TEXTLIST S1_Prompts
  0 = 'Waiting for Station 1 Clamp A1 Advance... Check Q1.0...' | German: 'S1_Prompts German 0' | French: 'S1_Prompts French 0' | 汉语: '汉语'
  1 = 'Waiting for Station 1 Clamp A1 Return... Check Q1.1...' | German: 'S1_Prompts German 1' | French: 'S1_Prompts French 1' | 汉语: '汉语'
  2 = 'Spare' | German: 'S1_Prompts German 2' | French: 'S1_Prompts French 2' | 汉语: '汉语'
  3 = 'Spare' | German: 'S1_Prompts German 3' | French: 'S1_Prompts French 3'
  4 = 'Spare' | German: 'S1_Prompts German 4' | French: 'S1_Prompts French 4'
  5 = 'Spare' | German: 'S1_Prompts German 5' | French: 'S1_Prompts French 5'
  6 = 'Spare' | German: 'S1_Prompts German 6' | French: 'S1_Prompts French 6'
  7 = 'Spare' | German: 'S1_Prompts German 7' | French: 'S1_Prompts French 7'
  8 = 'Spare' | German: 'S1_Prompts German 8' | French: 'S1_Prompts French 8'
  9 = 'Spare' | German: 'S1_Prompts German 9' | French: 'S1_Prompts French 9'
  10 = 'Waiting for Lock Cylinder A2 Lock... Check Q1.2...' | German: 'S1_Prompts German 10' | French: 'S1_Prompts French 10'
  11 = 'Waiting for Lock Cylinder A2 Unlock... Check Q1.3...' | German: 'S1_Prompts German 11' | French: 'S1_Prompts French 11'
  12 = 'Spare' | German: 'S1_Prompts German 12' | French: 'S1_Prompts French 12'
  13 = 'Spare' | German: 'S1_Prompts German 13' | French: 'S1_Prompts French 13'
  14 = 'Spare' | German: 'S1_Prompts German 14' | French: 'S1_Prompts French 14'
  15 = 'Spare' | German: 'S1_Prompts German 15' | French: 'S1_Prompts French 15'
  16 = 'Spare' | German: 'S1_Prompts German 16' | French: 'S1_Prompts French 16'
  17 = 'Spare' | German: 'S1_Prompts German 17' | French: 'S1_Prompts French 17'
  18 = 'Spare' | German: 'S1_Prompts German 18' | French: 'S1_Prompts French 18'
  19 = 'Spare' | German: 'S1_Prompts German 19' | French: 'S1_Prompts French 19'
  20 = 'Waiting for Urger Cylinder A3 Urge... Check Q1.4...' | German: 'S1_Prompts German 20' | French: 'S1_Prompts French 20'
  21 = 'Waiting for Urger Cylinder A3 Return... Check Q1.5...' | German: 'S1_Prompts German 21' | French: 'S1_Prompts French 21'
  22 = 'Spare' | German: 'S1_Prompts German 22' | French: 'S1_Prompts French 22'
  23 = 'Spare' | German: 'S1_Prompts German 23' | French: 'S1_Prompts French 23'
  24 = 'Spare' | German: 'S1_Prompts German 24' | French: 'S1_Prompts French 24'
  25 = 'Spare' | German: 'S1_Prompts German 25' | French: 'S1_Prompts French 25'
  26 = 'Spare' | German: 'S1_Prompts German 26' | French: 'S1_Prompts French 26'
  27 = 'Spare' | German: 'S1_Prompts German 27' | French: 'S1_Prompts French 27'
  28 = 'Spare' | German: 'S1_Prompts German 28' | French: 'S1_Prompts French 28'
  29 = 'Spare' | German: 'S1_Prompts German 29' | French: 'S1_Prompts French 29'
  30 = 'Waiting for Clamp Cylinder A1 Advance... Check Q1.0...' | German: 'S1_Prompts German 30' | French: 'S1_Prompts French 30'
  31 = 'Waiting for Clamp Cylinder A1 Return... Check Q1.1...' | German: 'S1_Prompts German 31' | French: 'S1_Prompts French 31'
  32 = 'Spare' | German: 'S1_Prompts German 32' | French: 'S1_Prompts French 32'
  33 = 'Spare' | German: 'S1_Prompts German 33' | French: 'S1_Prompts French 33'
  34 = 'Spare' | German: 'S1_Prompts German 34' | French: 'S1_Prompts French 34'
  35 = 'Spare' | German: 'S1_Prompts German 35' | French: 'S1_Prompts French 35'
  36 = 'Spare' | German: 'S1_Prompts German 36' | French: 'S1_Prompts French 36'
  37 = 'Spare' | German: 'S1_Prompts German 37' | French: 'S1_Prompts French 37'
  38 = 'Spare' | German: 'S1_Prompts German 38' | French: 'S1_Prompts French 38'
  39 = 'Spare' | German: 'S1_Prompts German 39' | French: 'S1_Prompts French 39'
  40 = 'Waiting for Clamp Cylinder A1 Advance... Check Q1.0...' | German: 'S1_Prompts German 40' | French: 'S1_Prompts French 40'
  41 = 'Waiting for Clamp Cylinder A1 Return... Check Q1.1...' | German: 'S1_Prompts German 41' | French: 'S1_Prompts French 41'
  42 = 'Spare' | German: 'S1_Prompts German 42' | French: 'S1_Prompts French 42'
  43 = 'Spare' | German: 'S1_Prompts German 43' | French: 'S1_Prompts French 43'
  44 = 'Spare' | German: 'S1_Prompts German 44' | French: 'S1_Prompts French 44'
  45 = 'Spare' | German: 'S1_Prompts German 45' | French: 'S1_Prompts French 45'
  46 = 'Spare' | German: 'S1_Prompts German 46' | French: 'S1_Prompts French 46'
  47 = 'Spare' | German: 'S1_Prompts German 47' | French: 'S1_Prompts French 47'
  48 = 'Spare' | German: 'S1_Prompts German 48' | French: 'S1_Prompts French 48'
  49 = 'Spare' | German: 'S1_Prompts German 49' | French: 'S1_Prompts French 49'
  50 = 'Waiting for Clamp Cylinder A1 Advance... Check Q1.0...' | German: 'S1_Prompts German 50' | French: 'S1_Prompts French 50'
  51 = 'Waiting for Clamp Cylinder A1 Return... Check Q1.1...' | German: 'S1_Prompts German 51' | French: 'S1_Prompts French 51'
  52 = 'Spare' | German: 'S1_Prompts German 52' | French: 'S1_Prompts French 52'
  53 = 'Spare' | German: 'S1_Prompts German 53' | French: 'S1_Prompts French 53'
  54 = 'Spare' | German: 'S1_Prompts German 54' | French: 'S1_Prompts French 54'
  55 = 'Spare' | German: 'S1_Prompts German 55' | French: 'S1_Prompts French 55'
  56 = 'Spare' | German: 'S1_Prompts German 56' | French: 'S1_Prompts French 56'
  57 = 'Spare' | German: 'S1_Prompts German 57' | French: 'S1_Prompts French 57'
  58 = 'Spare' | German: 'S1_Prompts German 58' | French: 'S1_Prompts French 58'
  59 = 'Spare' | German: 'S1_Prompts German 59' | French: 'S1_Prompts French 59'
  60 = 'Waiting for Clamp Cylinder A1 Advance... Check Q1.0...' | German: 'S1_Prompts German 60' | French: 'S1_Prompts French 60'
  61 = 'Waiting for Clamp Cylinder A1 Return... Check Q1.1...' | German: 'S1_Prompts German 61' | French: 'S1_Prompts French 61'
  62 = 'Spare' | German: 'S1_Prompts German 62' | French: 'S1_Prompts French 62'
  63 = 'Spare' | German: 'S1_Prompts German 63' | French: 'S1_Prompts French 63'
  64 = 'Spare' | German: 'S1_Prompts German 64' | French: 'S1_Prompts French 64'
  65 = 'Spare' | German: 'S1_Prompts German 65' | French: 'S1_Prompts French 65'
  66 = 'Spare' | German: 'S1_Prompts German 66' | French: 'S1_Prompts French 66'
  67 = 'Spare' | German: 'S1_Prompts German 67' | French: 'S1_Prompts French 67'
  68 = 'Spare' | German: 'S1_Prompts German 68' | French: 'S1_Prompts French 68'
  69 = 'Spare' | German: 'S1_Prompts German 69' | French: 'S1_Prompts French 69'
  70 = 'Waiting for Clamp Cylinder A1 Advance... Check Q1.0...' | German: 'S1_Prompts German 70' | French: 'S1_Prompts French 70'
  71 = 'Waiting for Clamp Cylinder A1 Return... Check Q1.1...' | German: 'S1_Prompts German 71' | French: 'S1_Prompts French 71'
  72 = 'Spare' | German: 'S1_Prompts German 72' | French: 'S1_Prompts French 72'
  73 = 'Spare' | German: 'S1_Prompts German 73' | French: 'S1_Prompts French 73'
  74 = 'Spare' | German: 'S1_Prompts German 74' | French: 'S1_Prompts French 74'
  75 = 'Spare' | German: 'S1_Prompts German 75' | French: 'S1_Prompts French 75'
  76 = 'Spare' | German: 'S1_Prompts German 76' | French: 'S1_Prompts French 76'
  77 = 'Spare' | German: 'S1_Prompts German 77' | French: 'S1_Prompts French 77'
  78 = 'Spare' | German: 'S1_Prompts German 78' | French: 'S1_Prompts French 78'
  79 = 'Spare' | German: 'S1_Prompts German 79' | French: 'S1_Prompts French 79'
  80 = 'Waiting for Clamp Cylinder A1 Advance... Check Q1.0...' | German: 'S1_Prompts German 80' | French: 'S1_Prompts French 80'
  81 = 'Waiting for Clamp Cylinder A1 Return... Check Q1.1...' | German: 'S1_Prompts German 81' | French: 'S1_Prompts French 81'
  82 = 'Spare' | German: 'S1_Prompts German 82' | French: 'S1_Prompts French 82'
  83 = 'Spare' | German: 'S1_Prompts German 83' | French: 'S1_Prompts French 83'
  84 = 'Spare' | German: 'S1_Prompts German 84' | French: 'S1_Prompts French 84'
  85 = 'Spare' | German: 'S1_Prompts German 85' | French: 'S1_Prompts French 85'
  86 = 'Spare' | German: 'S1_Prompts German 86' | French: 'S1_Prompts French 86'
  87 = 'Spare' | German: 'S1_Prompts German 87' | French: 'S1_Prompts French 87'
  88 = 'Spare' | German: 'S1_Prompts German 88' | French: 'S1_Prompts French 88'
  89 = 'Spare' | German: 'S1_Prompts German 89' | French: 'S1_Prompts French 89'
  90 = 'Waiting for Clamp Cylinder A1 Advance... Check Q1.0...' | German: 'S1_Prompts German 90' | French: 'S1_Prompts French 90'
  91 = 'Waiting for Clamp Cylinder A1 Return... Check Q1.1...' | German: 'S1_Prompts German 91' | French: 'S1_Prompts French 91'
  92 = 'Spare' | German: 'S1_Prompts German 92' | French: 'S1_Prompts French 92'
  93 = 'Spare' | German: 'S1_Prompts German 93' | French: 'S1_Prompts French 93'
  94 = 'Spare' | German: 'S1_Prompts German 94' | French: 'S1_Prompts French 94'
  95 = 'Spare' | German: 'S1_Prompts German 95' | French: 'S1_Prompts French 95'
  96 = 'Spare' | German: 'S1_Prompts German 96' | French: 'S1_Prompts French 96'
  97 = 'Spare' | German: 'S1_Prompts German 97' | French: 'S1_Prompts French 97'
  98 = 'Spare' | German: 'S1_Prompts German 98' | French: 'S1_Prompts French 98'
  99 = 'Spare' | German: 'S1_Prompts German 99' | French: 'S1_Prompts French 99'
  100 = 'Waiting for Clamp Cylinder A1 Advance... Check Q1.0...' | German: 'S1_Prompts German 100' | French: 'S1_Prompts French 100'
  101 = 'Waiting for Clamp Cylinder A1 Return... Check Q1.1...' | German: 'S1_Prompts German 101' | French: 'S1_Prompts French 101'
  102 = 'Spare' | German: 'S1_Prompts German 102' | French: 'S1_Prompts French 102'
  103 = 'Spare' | German: 'S1_Prompts German 103' | French: 'S1_Prompts French 103'
  104 = 'Spare' | German: 'S1_Prompts German 104' | French: 'S1_Prompts French 104'
  105 = 'Spare' | German: 'S1_Prompts German 105' | French: 'S1_Prompts French 105'
  106 = 'Spare' | German: 'S1_Prompts German 106' | French: 'S1_Prompts French 106'
  107 = 'Spare' | German: 'S1_Prompts German 107' | French: 'S1_Prompts French 107'
  108 = 'Spare' | German: 'S1_Prompts German 108' | French: 'S1_Prompts French 108'
  109 = 'Spare' | German: 'S1_Prompts German 109' | French: 'S1_Prompts French 109'
  110 = 'Waiting for Clamp Cylinder A1 Advance... Check Q1.0...' | German: 'S1_Prompts German 110' | French: 'S1_Prompts French 110'
  111 = 'Waiting for Clamp Cylinder A1 Return... Check Q1.1...' | German: 'S1_Prompts German 111' | French: 'S1_Prompts French 111'
  112 = 'Spare' | German: 'S1_Prompts German 112' | French: 'S1_Prompts French 112'
  113 = 'Spare' | German: 'S1_Prompts German 113' | French: 'S1_Prompts French 113'
  114 = 'Spare' | German: 'S1_Prompts German 114' | French: 'S1_Prompts French 114'
  115 = 'Spare' | German: 'S1_Prompts German 115' | French: 'S1_Prompts French 115'
  116 = 'Spare' | German: 'S1_Prompts German 116' | French: 'S1_Prompts French 116'
  117 = 'Spare' | German: 'S1_Prompts German 117' | French: 'S1_Prompts French 117'
  118 = 'Spare' | German: 'S1_Prompts German 118' | French: 'S1_Prompts French 118'
  119 = 'Spare' | German: 'S1_Prompts German 119' | French: 'S1_Prompts French 119'
  120 = 'Waiting for Clamp Cylinder A1 Advance... Check Q1.0...' | German: 'S1_Prompts German 120' | French: 'S1_Prompts French 120'
  121 = 'Waiting for Clamp Cylinder A1 Return... Check Q1.1...' | German: 'S1_Prompts German 121' | French: 'S1_Prompts French 121'
  122 = 'Spare' | German: 'S1_Prompts German 122' | French: 'S1_Prompts French 122'
  123 = 'Spare' | German: 'S1_Prompts German 123' | French: 'S1_Prompts French 123'
  124 = 'Spare' | German: 'S1_Prompts German 124' | French: 'S1_Prompts French 124'
  125 = 'Spare' | German: 'S1_Prompts German 125' | French: 'S1_Prompts French 125'
  126 = 'Spare' | German: 'S1_Prompts German 126' | French: 'S1_Prompts French 126'
  127 = 'Spare' | German: 'S1_Prompts German 127' | French: 'S1_Prompts French 127'
  128 = 'Spare' | German: 'S1_Prompts German 128' | French: 'S1_Prompts French 128'
  129 = 'Spare' | German: 'S1_Prompts German 129' | French: 'S1_Prompts French 129'
  130 = 'Waiting for Clamp Cylinder A1 Advance... Check Q1.0...' | German: 'S1_Prompts German 130' | French: 'S1_Prompts French 130'
  131 = 'Waiting for Clamp Cylinder A1 Return... Check Q1.1...' | German: 'S1_Prompts German 131' | French: 'S1_Prompts French 131'
  132 = 'Spare' | German: 'S1_Prompts German 132' | French: 'S1_Prompts French 132'
  133 = 'Spare' | German: 'S1_Prompts German 133' | French: 'S1_Prompts French 133'
  134 = 'Spare' | German: 'S1_Prompts German 134' | French: 'S1_Prompts French 134'
  135 = 'Spare' | German: 'S1_Prompts German 135' | French: 'S1_Prompts French 135'
  136 = 'Spare' | German: 'S1_Prompts German 136' | French: 'S1_Prompts French 136'
  137 = 'Spare' | German: 'S1_Prompts German 137' | French: 'S1_Prompts French 137'
  138 = 'Spare' | German: 'S1_Prompts German 138' | French: 'S1_Prompts French 138'
  139 = 'Spare' | German: 'S1_Prompts German 139' | French: 'S1_Prompts French 139'
  140 = 'Waiting for Clamp Cylinder A1 Advance... Check Q1.0...' | German: 'S1_Prompts German 140' | French: 'S1_Prompts French 140'
  141 = 'Waiting for Clamp Cylinder A1 Return... Check Q1.1...' | German: 'S1_Prompts German 141' | French: 'S1_Prompts French 141'
  142 = 'Spare' | German: 'S1_Prompts German 142' | French: 'S1_Prompts French 142'
  143 = 'Spare' | German: 'S1_Prompts German 143' | French: 'S1_Prompts French 143'
  144 = 'Spare' | German: 'S1_Prompts German 144' | French: 'S1_Prompts French 144'
  145 = 'Spare' | German: 'S1_Prompts German 145' | French: 'S1_Prompts French 145'
  146 = 'Spare' | German: 'S1_Prompts German 146' | French: 'S1_Prompts French 146'
  147 = 'Spare' | German: 'S1_Prompts German 147' | French: 'S1_Prompts French 147'
  148 = 'Spare' | German: 'S1_Prompts German 148' | French: 'S1_Prompts French 148'
  149 = 'Spare' | German: 'S1_Prompts German 149' | French: 'S1_Prompts French 149'
  150 = 'Waiting for Clamp Cylinder A1 Advance... Check Q1.0...' | German: 'S1_Prompts German 150' | French: 'S1_Prompts French 150'
  151 = 'Waiting for Clamp Cylinder A1 Return... Check Q1.1...' | German: 'S1_Prompts German 151' | French: 'S1_Prompts French 151'
  152 = 'Spare' | German: 'S1_Prompts German 152' | French: 'S1_Prompts French 152'
  153 = 'Spare' | German: 'S1_Prompts German 153' | French: 'S1_Prompts French 153'
  154 = 'Spare' | German: 'S1_Prompts German 154' | French: 'S1_Prompts French 154'
  155 = 'Spare' | German: 'S1_Prompts German 155' | French: 'S1_Prompts French 155'
  156 = 'Spare' | German: 'S1_Prompts German 156' | French: 'S1_Prompts French 156'
  157 = 'Spare' | German: 'S1_Prompts German 157' | French: 'S1_Prompts French 157'
  158 = 'Spare' | German: 'S1_Prompts German 158' | French: 'S1_Prompts French 158'
  159 = 'Spare' | German: 'S1_Prompts German 159' | French: 'S1_Prompts French 159'
  160 = 'Waiting for Clamp Cylinder A1 Advance... Check Q1.0...' | German: 'S1_Prompts German 160' | French: 'S1_Prompts French 160'
  161 = 'Waiting for Clamp Cylinder A1 Return... Check Q1.1...' | German: 'S1_Prompts German 161' | French: 'S1_Prompts French 161'
  162 = 'Spare' | German: 'S1_Prompts German 162' | French: 'S1_Prompts French 162'
  163 = 'Spare' | German: 'S1_Prompts German 163' | French: 'S1_Prompts French 163'
  164 = 'Spare' | German: 'S1_Prompts German 164' | French: 'S1_Prompts French 164'
  165 = 'Spare' | German: 'S1_Prompts German 165' | French: 'S1_Prompts French 165'
  166 = 'Spare' | German: 'S1_Prompts German 166' | French: 'S1_Prompts French 166'
  167 = 'Spare' | German: 'S1_Prompts German 167' | French: 'S1_Prompts French 167'
  168 = 'Spare' | German: 'S1_Prompts German 168' | French: 'S1_Prompts French 168'
  169 = 'Spare' | German: 'S1_Prompts German 169' | French: 'S1_Prompts French 169'
  170 = 'Waiting for Clamp Cylinder A1 Advance... Check Q1.0...' | German: 'S1_Prompts German 170' | French: 'S1_Prompts French 170'
  171 = 'Waiting for Clamp Cylinder A1 Return... Check Q1.1...' | German: 'S1_Prompts German 171' | French: 'S1_Prompts French 171'
  172 = 'Spare' | German: 'S1_Prompts German 172' | French: 'S1_Prompts French 172'
  173 = 'Spare' | German: 'S1_Prompts German 173' | French: 'S1_Prompts French 173'
  174 = 'Spare' | German: 'S1_Prompts German 174' | French: 'S1_Prompts French 174'
  175 = 'Spare' | German: 'S1_Prompts German 175' | French: 'S1_Prompts French 175'
  176 = 'Spare' | German: 'S1_Prompts German 176' | French: 'S1_Prompts French 176'
  177 = 'Spare' | German: 'S1_Prompts German 177' | French: 'S1_Prompts French 177'
  178 = 'Spare' | German: 'S1_Prompts German 178' | French: 'S1_Prompts French 178'
  179 = 'Spare' | German: 'S1_Prompts German 179' | French: 'S1_Prompts French 179'
  180 = 'Waiting for Clamp Cylinder A1 Advance... Check Q1.0...' | German: 'S1_Prompts German 180' | French: 'S1_Prompts French 180'
  181 = 'Waiting for Clamp Cylinder A1 Return... Check Q1.1...' | German: 'S1_Prompts German 181' | French: 'S1_Prompts French 181'
  182 = 'Spare' | German: 'S1_Prompts German 182' | French: 'S1_Prompts French 182'
  183 = 'Spare' | German: 'S1_Prompts German 183' | French: 'S1_Prompts French 183'
  184 = 'Spare' | German: 'S1_Prompts German 184' | French: 'S1_Prompts French 184'
  185 = 'Spare' | German: 'S1_Prompts German 185' | French: 'S1_Prompts French 185'
  186 = 'Spare' | German: 'S1_Prompts German 186' | French: 'S1_Prompts French 186'
  187 = 'Spare' | German: 'S1_Prompts German 187' | French: 'S1_Prompts French 187'
  188 = 'Spare' | German: 'S1_Prompts German 188' | French: 'S1_Prompts French 188'
  189 = 'Spare' | German: 'S1_Prompts German 189' | French: 'S1_Prompts French 189'
  190 = 'Waiting for Clamp Cylinder A1 Advance... Check Q1.0...' | German: 'S1_Prompts German 190' | French: 'S1_Prompts French 190'
  191 = 'Waiting for Clamp Cylinder A1 Return... Check Q1.1...' | German: 'S1_Prompts German 191' | French: 'S1_Prompts French 191'
  192 = 'Spare' | German: 'S1_Prompts German 192' | French: 'S1_Prompts French 192'
  193 = 'Spare' | German: 'S1_Prompts German 193' | French: 'S1_Prompts French 193'
  194 = 'Spare' | German: 'S1_Prompts German 194' | French: 'S1_Prompts French 194'
  195 = 'Spare' | German: 'S1_Prompts German 195' | French: 'S1_Prompts French 195'
  196 = 'Spare' | German: 'S1_Prompts German 196' | French: 'S1_Prompts French 196'
  197 = 'Spare' | German: 'S1_Prompts German 197' | French: 'S1_Prompts French 197'
  198 = 'Spare' | German: 'S1_Prompts German 198' | French: 'S1_Prompts French 198'
  199 = 'Spare' | German: 'S1_Prompts German 199' | French: 'S1_Prompts French 199'
  200 = 'Waiting for Clamp Cylinder A1 Advance... Check Q1.0...' | German: 'S1_Prompts German 200' | French: 'S1_Prompts French 200'
  201 = 'Waiting for Clamp Cylinder A1 Return... Check Q1.1...' | German: 'S1_Prompts German 201' | French: 'S1_Prompts French 201'
  202 = 'Spare' | German: 'S1_Prompts German 202' | French: 'S1_Prompts French 202'
  203 = 'Spare' | German: 'S1_Prompts German 203' | French: 'S1_Prompts French 203'
  204 = 'Spare' | German: 'S1_Prompts German 204' | French: 'S1_Prompts French 204'
  205 = 'Spare' | German: 'S1_Prompts German 205' | French: 'S1_Prompts French 205'
  206 = 'Spare' | German: 'S1_Prompts German 206' | French: 'S1_Prompts French 206'
  207 = 'Spare' | German: 'S1_Prompts German 207' | French: 'S1_Prompts French 207'
  208 = 'Spare' | German: 'S1_Prompts German 208' | French: 'S1_Prompts French 208'
  209 = 'Spare' | German: 'S1_Prompts German 209' | French: 'S1_Prompts French 209'
  210 = 'Waiting for Clamp Cylinder A1 Advance... Check Q1.0...' | German: 'S1_Prompts German 210' | French: 'S1_Prompts French 210'
  211 = 'Waiting for Clamp Cylinder A1 Return... Check Q1.1...' | German: 'S1_Prompts German 211' | French: 'S1_Prompts French 211'
  212 = 'Spare' | German: 'S1_Prompts German 212' | French: 'S1_Prompts French 212'
  213 = 'Spare' | German: 'S1_Prompts German 213' | French: 'S1_Prompts French 213'
  214 = 'Spare' | German: 'S1_Prompts German 214' | French: 'S1_Prompts French 214'
  215 = 'Spare' | German: 'S1_Prompts German 215' | French: 'S1_Prompts French 215'
  216 = 'Spare' | German: 'S1_Prompts German 216' | French: 'S1_Prompts French 216'
  217 = 'Spare' | German: 'S1_Prompts German 217' | French: 'S1_Prompts French 217'
  218 = 'Spare' | German: 'S1_Prompts German 218' | French: 'S1_Prompts French 218'
  219 = 'Spare' | German: 'S1_Prompts German 219' | French: 'S1_Prompts French 219'
  220 = 'Waiting for Clamp Cylinder A1 Advance... Check Q1.0...' | German: 'S1_Prompts German 220' | French: 'S1_Prompts French 220'
  221 = 'Waiting for Clamp Cylinder A1 Return... Check Q1.1...' | German: 'S1_Prompts German 221' | French: 'S1_Prompts French 221'
  222 = 'Spare' | German: 'S1_Prompts German 222' | French: 'S1_Prompts French 222'
  223 = 'Spare' | German: 'S1_Prompts German 223' | French: 'S1_Prompts French 223'
  224 = 'Spare' | German: 'S1_Prompts German 224' | French: 'S1_Prompts French 224'
  225 = 'Spare' | German: 'S1_Prompts German 225' | French: 'S1_Prompts French 225'
  226 = 'Spare' | German: 'S1_Prompts German 226' | French: 'S1_Prompts French 226'
  227 = 'Spare' | German: 'S1_Prompts German 227' | French: 'S1_Prompts French 227'
  228 = 'Spare' | German: 'S1_Prompts German 228' | French: 'S1_Prompts French 228'
  229 = 'Spare' | German: 'S1_Prompts German 229' | French: 'S1_Prompts French 229'
  230 = 'Waiting for Clamp Cylinder A1 Advance... Check Q1.0...' | German: 'S1_Prompts German 230' | French: 'S1_Prompts French 230'
  231 = 'Waiting for Clamp Cylinder A1 Return... Check Q1.1...' | German: 'S1_Prompts German 231' | French: 'S1_Prompts French 231'
  232 = 'Spare' | German: 'S1_Prompts German 232' | French: 'S1_Prompts French 232'
  233 = 'Spare' | German: 'S1_Prompts German 233' | French: 'S1_Prompts French 233'
  234 = 'Spare' | German: 'S1_Prompts German 234' | French: 'S1_Prompts French 234'
  235 = 'Spare' | German: 'S1_Prompts German 235' | French: 'S1_Prompts French 235'
  236 = 'Spare' | German: 'S1_Prompts German 236' | French: 'S1_Prompts French 236'
  237 = 'Spare' | German: 'S1_Prompts German 237' | French: 'S1_Prompts French 237'
  238 = 'Spare' | German: 'S1_Prompts German 238' | French: 'S1_Prompts French 238'
  239 = 'Spare' | German: 'S1_Prompts German 239' | French: 'S1_Prompts French 239'
  240 = 'Waiting for Clamp Cylinder A1 Advance... Check Q1.0...' | German: 'S1_Prompts German 240' | French: 'S1_Prompts French 240'
  241 = 'Waiting for Clamp Cylinder A1 Return... Check Q1.1...' | German: 'S1_Prompts German 241' | French: 'S1_Prompts French 241'
  242 = 'Spare' | German: 'S1_Prompts German 242' | French: 'S1_Prompts French 242'
  243 = 'Spare' | German: 'S1_Prompts German 243' | French: 'S1_Prompts French 243'
  244 = 'Spare' | German: 'S1_Prompts German 244' | French: 'S1_Prompts French 244'
  245 = 'Spare' | German: 'S1_Prompts German 245' | French: 'S1_Prompts French 245'
  246 = 'Spare' | German: 'S1_Prompts German 246' | French: 'S1_Prompts French 246'
  247 = 'Spare' | German: 'S1_Prompts German 247' | French: 'S1_Prompts French 247'
  248 = 'Spare' | German: 'S1_Prompts German 248' | French: 'S1_Prompts French 248'
  249 = 'Spare' | German: 'S1_Prompts German 249' | French: 'S1_Prompts French 249'
  250 = 'Waiting for Clamp Cylinder A1 Advance... Check Q1.0...' | German: 'S1_Prompts German 250' | French: 'S1_Prompts French 250'
  251 = 'Waiting for Clamp Cylinder A1 Return... Check Q1.1...' | German: 'S1_Prompts German 251' | French: 'S1_Prompts French 251'
  252 = 'Spare' | German: 'S1_Prompts German 252' | French: 'S1_Prompts French 252'
  253 = 'Spare' | German: 'S1_Prompts German 253' | French: 'S1_Prompts French 253'
  254 = 'Spare' | German: 'S1_Prompts German 254' | French: 'S1_Prompts French 254'
  255 = 'Spare' | German: 'S1_Prompts German 255' | French: 'S1_Prompts French 255'
  256 = 'Spare' | German: 'S1_Prompts German 256' | French: 'S1_Prompts French 256'
  257 = 'Spare' | German: 'S1_Prompts German 257' | French: 'S1_Prompts French 257'
  258 = 'Spare' | German: 'S1_Prompts German 258' | French: 'S1_Prompts French 258'
  259 = 'Spare' | German: 'S1_Prompts German 259' | French: 'S1_Prompts French 259'
  260 = 'Waiting for Clamp Cylinder A1 Advance... Check Q1.0...' | German: 'S1_Prompts German 260' | French: 'S1_Prompts French 260'
  261 = 'Waiting for Clamp Cylinder A1 Return... Check Q1.1...' | German: 'S1_Prompts German 261' | French: 'S1_Prompts French 261'
  262 = 'Spare' | German: 'S1_Prompts German 262' | French: 'S1_Prompts French 262'
  263 = 'Spare' | German: 'S1_Prompts German 263' | French: 'S1_Prompts French 263'
  264 = 'Spare' | German: 'S1_Prompts German 264' | French: 'S1_Prompts French 264'
  265 = 'Spare' | German: 'S1_Prompts German 265' | French: 'S1_Prompts French 265'
  266 = 'Spare' | German: 'S1_Prompts German 266' | French: 'S1_Prompts French 266'
  267 = 'Spare' | German: 'S1_Prompts German 267' | French: 'S1_Prompts French 267'
  268 = 'Spare' | German: 'S1_Prompts German 268' | French: 'S1_Prompts French 268'
  269 = 'Spare' | German: 'S1_Prompts German 269' | French: 'S1_Prompts French 269'
  270 = 'Waiting for Clamp Cylinder A1 Advance... Check Q1.0...' | German: 'S1_Prompts German 270' | French: 'S1_Prompts French 270'
  271 = 'Waiting for Clamp Cylinder A1 Return... Check Q1.1...' | German: 'S1_Prompts German 271' | French: 'S1_Prompts French 271'
  272 = 'Spare' | German: 'S1_Prompts German 272' | French: 'S1_Prompts French 272'
  273 = 'Spare' | German: 'S1_Prompts German 273' | French: 'S1_Prompts French 273'
  274 = 'Spare' | German: 'S1_Prompts German 274' | French: 'S1_Prompts French 274'
  275 = 'Spare' | German: 'S1_Prompts German 275' | French: 'S1_Prompts French 275'
  276 = 'Spare' | German: 'S1_Prompts German 276' | French: 'S1_Prompts French 276'
  277 = 'Spare' | German: 'S1_Prompts German 277' | French: 'S1_Prompts French 277'
  278 = 'Spare' | German: 'S1_Prompts German 278' | French: 'S1_Prompts French 278'
  279 = 'Spare' | German: 'S1_Prompts German 279' | French: 'S1_Prompts French 279'
  280 = 'Waiting for Clamp Cylinder A1 Advance... Check Q1.0...' | German: 'S1_Prompts German 280' | French: 'S1_Prompts French 280'
  281 = 'Waiting for Clamp Cylinder A1 Return... Check Q1.1...' | German: 'S1_Prompts German 281' | French: 'S1_Prompts French 281'
  282 = 'Spare' | German: 'S1_Prompts German 282' | French: 'S1_Prompts French 282'
  283 = 'Spare' | German: 'S1_Prompts German 283' | French: 'S1_Prompts French 283'
  284 = 'Spare' | German: 'S1_Prompts German 284' | French: 'S1_Prompts French 284'
  285 = 'Spare' | German: 'S1_Prompts German 285' | French: 'S1_Prompts French 285'
  286 = 'Spare' | German: 'S1_Prompts German 286' | French: 'S1_Prompts French 286'
  287 = 'Spare' | German: 'S1_Prompts German 287' | French: 'S1_Prompts French 287'
  288 = 'Spare' | German: 'S1_Prompts German 288' | French: 'S1_Prompts French 288'
  289 = 'Spare' | German: 'S1_Prompts German 289' | French: 'S1_Prompts French 289'
  290 = 'Waiting for Clamp Cylinder A1 Advance... Check Q1.0...' | German: 'S1_Prompts German 290' | French: 'S1_Prompts French 290'
  291 = 'Waiting for Clamp Cylinder A1 Return... Check Q1.1...' | German: 'S1_Prompts German 291' | French: 'S1_Prompts French 291'
  292 = 'Spare' | German: 'S1_Prompts German 292' | French: 'S1_Prompts French 292'
  293 = 'Spare' | German: 'S1_Prompts German 293' | French: 'S1_Prompts French 293'
  294 = 'Spare' | German: 'S1_Prompts German 294' | French: 'S1_Prompts French 294'
  295 = 'Spare' | German: 'S1_Prompts German 295' | French: 'S1_Prompts French 295'
  296 = 'Spare' | German: 'S1_Prompts German 296' | French: 'S1_Prompts French 296'
  297 = 'Spare' | German: 'S1_Prompts German 297' | French: 'S1_Prompts French 297'
  298 = 'Spare' | German: 'S1_Prompts German 298' | French: 'S1_Prompts French 298'
  299 = 'Spare' | German: 'S1_Prompts German 299' | French: 'S1_Prompts French 299'
  300 = 'Waiting for Clamp Cylinder A1 Advance... Check Q1.0...' | German: 'S1_Prompts German 300' | French: 'S1_Prompts French 300'
  301 = 'Waiting for Clamp Cylinder A1 Return... Check Q1.1...' | German: 'S1_Prompts German 301' | French: 'S1_Prompts French 301'
  302 = 'Spare' | German: 'S1_Prompts German 302' | French: 'S1_Prompts French 302'
  303 = 'Spare' | German: 'S1_Prompts German 303' | French: 'S1_Prompts French 303'
  304 = 'Spare' | German: 'S1_Prompts German 304' | French: 'S1_Prompts French 304'
  305 = 'Spare' | German: 'S1_Prompts German 305' | French: 'S1_Prompts French 305'
  306 = 'Spare' | German: 'S1_Prompts German 306' | French: 'S1_Prompts French 306'
  307 = 'Spare' | German: 'S1_Prompts German 307' | French: 'S1_Prompts French 307'
  308 = 'Spare' | German: 'S1_Prompts German 308' | French: 'S1_Prompts French 308'
  309 = 'Spare' | German: 'S1_Prompts German 309' | French: 'S1_Prompts French 309'
  310 = 'Waiting for Clamp Cylinder A1 Advance... Check Q1.0...' | German: 'S1_Prompts German 310' | French: 'S1_Prompts French 310'
  311 = 'Waiting for Clamp Cylinder A1 Return... Check Q1.1...' | German: 'S1_Prompts German 311' | French: 'S1_Prompts French 311'
  312 = 'Spare' | German: 'S1_Prompts German 312' | French: 'S1_Prompts French 312'
  313 = 'Spare' | German: 'S1_Prompts German 313' | French: 'S1_Prompts French 313'
  314 = 'Spare' | German: 'S1_Prompts German 314' | French: 'S1_Prompts French 314'
  315 = 'Spare' | German: 'S1_Prompts German 315' | French: 'S1_Prompts French 315'
  316 = 'Spare' | German: 'S1_Prompts German 316' | French: 'S1_Prompts French 316'
  317 = 'Spare' | German: 'S1_Prompts German 317' | French: 'S1_Prompts French 317'
  318 = 'Spare' | German: 'S1_Prompts German 318' | French: 'S1_Prompts French 318'
  319 = 'Spare' | German: 'S1_Prompts German 319' | French: 'S1_Prompts French 319'
  320 = 'Waiting for Clamp Cylinder A1 Advance... Check Q1.0...' | German: 'S1_Prompts German 320' | French: 'S1_Prompts French 320'
  321 = 'Waiting for Clamp Cylinder A1 Return... Check Q1.1...' | German: 'S1_Prompts German 321' | French: 'S1_Prompts French 321'
  322 = 'Spare' | German: 'S1_Prompts German 322' | French: 'S1_Prompts French 322'
  323 = 'Spare' | German: 'S1_Prompts German 323' | French: 'S1_Prompts French 323'
  324 = 'Spare' | German: 'S1_Prompts German 324' | French: 'S1_Prompts French 324'
  325 = 'Spare' | German: 'S1_Prompts German 325' | French: 'S1_Prompts French 325'
  326 = 'Spare' | German: 'S1_Prompts German 326' | French: 'S1_Prompts French 326'
  327 = 'Spare' | German: 'S1_Prompts German 327' | French: 'S1_Prompts French 327'
  328 = 'Spare' | German: 'S1_Prompts German 328' | French: 'S1_Prompts French 328'
  329 = 'Spare' | German: 'S1_Prompts German 329' | French: 'S1_Prompts French 329'
  330 = 'Waiting for Clamp Cylinder A1 Advance... Check Q1.0...' | German: 'S1_Prompts German 330' | French: 'S1_Prompts French 330'
  331 = 'Waiting for Clamp Cylinder A1 Return... Check Q1.1...' | German: 'S1_Prompts German 331' | French: 'S1_Prompts French 331'
  332 = 'Spare' | German: 'S1_Prompts German 332' | French: 'S1_Prompts French 332'
  333 = 'Spare' | German: 'S1_Prompts German 333' | French: 'S1_Prompts French 333'
  334 = 'Spare' | German: 'S1_Prompts German 334' | French: 'S1_Prompts French 334'
  335 = 'Spare' | German: 'S1_Prompts German 335' | French: 'S1_Prompts French 335'
  336 = 'Spare' | German: 'S1_Prompts German 336' | French: 'S1_Prompts French 336'
  337 = 'Spare' | German: 'S1_Prompts German 337' | French: 'S1_Prompts French 337'
  338 = 'Spare' | German: 'S1_Prompts German 338' | French: 'S1_Prompts French 338'
  339 = 'Spare' | German: 'S1_Prompts German 339' | French: 'S1_Prompts French 339'
  340 = 'Waiting for Clamp Cylinder A1 Advance... Check Q1.0...' | German: 'S1_Prompts German 340' | French: 'S1_Prompts French 340'
  341 = 'Waiting for Clamp Cylinder A1 Return... Check Q1.1...' | German: 'S1_Prompts German 341' | French: 'S1_Prompts French 341'
  342 = 'Spare' | German: 'S1_Prompts German 342' | French: 'S1_Prompts French 342'
  343 = 'Spare' | German: 'S1_Prompts German 343' | French: 'S1_Prompts French 343'
  344 = 'Spare' | German: 'S1_Prompts German 344' | French: 'S1_Prompts French 344'
  345 = 'Spare' | German: 'S1_Prompts German 345' | French: 'S1_Prompts French 345'
  346 = 'Spare' | German: 'S1_Prompts German 346' | French: 'S1_Prompts French 346'
  347 = 'Spare' | German: 'S1_Prompts German 347' | French: 'S1_Prompts French 347'
  348 = 'Spare' | German: 'S1_Prompts German 348' | French: 'S1_Prompts French 348'
  349 = 'Spare' | German: 'S1_Prompts German 349' | French: 'S1_Prompts French 349'
  350 = 'Waiting for Clamp Cylinder A1 Advance... Check Q1.0...' | German: 'S1_Prompts German 350' | French: 'S1_Prompts French 350'
  351 = 'Waiting for Clamp Cylinder A1 Return... Check Q1.1...' | German: 'S1_Prompts German 351' | French: 'S1_Prompts French 351'
  352 = 'Spare' | German: 'S1_Prompts German 352' | French: 'S1_Prompts French 352'
  353 = 'Spare' | German: 'S1_Prompts German 353' | French: 'S1_Prompts French 353'
  354 = 'Spare' | German: 'S1_Prompts German 354' | French: 'S1_Prompts French 354'
  355 = 'Spare' | German: 'S1_Prompts German 355' | French: 'S1_Prompts French 355'
  356 = 'Spare' | German: 'S1_Prompts German 356' | French: 'S1_Prompts French 356'
  357 = 'Spare' | German: 'S1_Prompts German 357' | French: 'S1_Prompts French 357'
  358 = 'Spare' | German: 'S1_Prompts German 358' | French: 'S1_Prompts French 358'
  359 = 'Spare' | German: 'S1_Prompts German 359' | French: 'S1_Prompts French 359'
  360 = 'Waiting for Clamp Cylinder A1 Advance... Check Q1.0...' | German: 'S1_Prompts German 360' | French: 'S1_Prompts French 360'
  361 = 'Waiting for Clamp Cylinder A1 Return... Check Q1.1...' | German: 'S1_Prompts German 361' | French: 'S1_Prompts French 361'
  362 = 'Spare' | German: 'S1_Prompts German 362' | French: 'S1_Prompts French 362'
  363 = 'Spare' | German: 'S1_Prompts German 363' | French: 'S1_Prompts French 363'
  364 = 'Spare' | German: 'S1_Prompts German 364' | French: 'S1_Prompts French 364'
  365 = 'Spare' | German: 'S1_Prompts German 365' | French: 'S1_Prompts French 365'
  366 = 'Spare' | German: 'S1_Prompts German 366' | French: 'S1_Prompts French 366'
  367 = 'Spare' | German: 'S1_Prompts German 367' | French: 'S1_Prompts French 367'
  368 = 'Spare' | German: 'S1_Prompts German 368' | French: 'S1_Prompts French 368'
  369 = 'Spare' | German: 'S1_Prompts German 369' | French: 'S1_Prompts French 369'
  370 = 'Waiting for Clamp Cylinder A1 Advance... Check Q1.0...' | German: 'S1_Prompts German 370' | French: 'S1_Prompts French 370'
  371 = 'Waiting for Clamp Cylinder A1 Return... Check Q1.1...' | German: 'S1_Prompts German 371' | French: 'S1_Prompts French 371'
  372 = 'Spare' | German: 'S1_Prompts German 372' | French: 'S1_Prompts French 372'
  373 = 'Spare' | German: 'S1_Prompts German 373' | French: 'S1_Prompts French 373'
  374 = 'Spare' | German: 'S1_Prompts German 374' | French: 'S1_Prompts French 374'
  375 = 'Spare' | German: 'S1_Prompts German 375' | French: 'S1_Prompts French 375'
  376 = 'Spare' | German: 'S1_Prompts German 376' | French: 'S1_Prompts French 376'
  377 = 'Spare' | German: 'S1_Prompts German 377' | French: 'S1_Prompts French 377'
  378 = 'Spare' | German: 'S1_Prompts German 378' | French: 'S1_Prompts French 378'
  379 = 'Spare' | German: 'S1_Prompts German 379' | French: 'S1_Prompts French 379'
  380 = 'Waiting for Clamp Cylinder A1 Advance... Check Q1.0...' | German: 'S1_Prompts German 380' | French: 'S1_Prompts French 380'
  381 = 'Waiting for Clamp Cylinder A1 Return... Check Q1.1...' | German: 'S1_Prompts German 381' | French: 'S1_Prompts French 381'
  382 = 'Spare' | German: 'S1_Prompts German 382' | French: 'S1_Prompts French 382'
  383 = 'Spare' | German: 'S1_Prompts German 383' | French: 'S1_Prompts French 383'
  384 = 'Spare' | German: 'S1_Prompts German 384' | French: 'S1_Prompts French 384'
  385 = 'Spare' | German: 'S1_Prompts German 385' | French: 'S1_Prompts French 385'
  386 = 'Spare' | German: 'S1_Prompts German 386' | French: 'S1_Prompts French 386'
  387 = 'Spare' | German: 'S1_Prompts German 387' | French: 'S1_Prompts French 387'
  388 = 'Spare' | German: 'S1_Prompts German 388' | French: 'S1_Prompts French 388'
  389 = 'Spare' | German: 'S1_Prompts German 389' | French: 'S1_Prompts French 389'
  390 = 'Waiting for Clamp Cylinder A1 Advance... Check Q1.0...' | German: 'S1_Prompts German 390' | French: 'S1_Prompts French 390'
  391 = 'Waiting for Clamp Cylinder A1 Return... Check Q1.1...' | German: 'S1_Prompts German 391' | French: 'S1_Prompts French 391'
  392 = 'Spare' | German: 'S1_Prompts German 392' | French: 'S1_Prompts French 392'
  393 = 'Spare' | German: 'S1_Prompts German 393' | French: 'S1_Prompts French 393'
  394 = 'Spare' | German: 'S1_Prompts German 394' | French: 'S1_Prompts French 394'
  395 = 'Spare' | German: 'S1_Prompts German 395' | French: 'S1_Prompts French 395'
  396 = 'Spare' | German: 'S1_Prompts German 396' | French: 'S1_Prompts French 396'
  397 = 'Spare' | German: 'S1_Prompts German 397' | French: 'S1_Prompts French 397'
  398 = 'Spare' | German: 'S1_Prompts German 398' | French: 'S1_Prompts French 398'
  399 = 'Spare' | German: 'S1_Prompts German 399' | French: 'S1_Prompts French 399'
  400 = 'Waiting for Clamp Cylinder A1 Advance... Check Q1.0...' | German: 'S1_Prompts German 400' | French: 'S1_Prompts French 400'
  401 = 'Waiting for Clamp Cylinder A1 Return... Check Q1.1...' | German: 'S1_Prompts German 401' | French: 'S1_Prompts French 401'
  402 = 'Spare' | German: 'S1_Prompts German 402' | French: 'S1_Prompts French 402'
  403 = 'Spare' | German: 'S1_Prompts German 403' | French: 'S1_Prompts French 403'
  404 = 'Spare' | German: 'S1_Prompts German 404' | French: 'S1_Prompts French 404'
  405 = 'Spare' | German: 'S1_Prompts German 405' | French: 'S1_Prompts French 405'
  406 = 'Spare' | German: 'S1_Prompts German 406' | French: 'S1_Prompts French 406'
  407 = 'Spare' | German: 'S1_Prompts German 407' | French: 'S1_Prompts French 407'
  408 = 'Spare' | German: 'S1_Prompts German 408' | French: 'S1_Prompts French 408'
  409 = 'Spare' | German: 'S1_Prompts German 409' | French: 'S1_Prompts French 409'
  410 = 'Waiting for Clamp Cylinder A1 Advance... Check Q1.0...' | German: 'S1_Prompts German 410' | French: 'S1_Prompts French 410'
  411 = 'Waiting for Clamp Cylinder A1 Return... Check Q1.1...' | German: 'S1_Prompts German 411' | French: 'S1_Prompts French 411'
  412 = 'Spare' | German: 'S1_Prompts German 412' | French: 'S1_Prompts French 412'
  413 = 'Spare' | German: 'S1_Prompts German 413' | French: 'S1_Prompts French 413'
  414 = 'Spare' | German: 'S1_Prompts German 414' | French: 'S1_Prompts French 414'
  415 = 'Spare' | German: 'S1_Prompts German 415' | French: 'S1_Prompts French 415'
  416 = 'Spare' | German: 'S1_Prompts German 416' | French: 'S1_Prompts French 416'
  417 = 'Spare' | German: 'S1_Prompts German 417' | French: 'S1_Prompts French 417'
  418 = 'Spare' | German: 'S1_Prompts German 418' | French: 'S1_Prompts French 418'
  419 = 'Spare' | German: 'S1_Prompts German 419' | French: 'S1_Prompts French 419'
  420 = 'Waiting for Clamp Cylinder A1 Advance... Check Q1.0...' | German: 'S1_Prompts German 420' | French: 'S1_Prompts French 420'
  421 = 'Waiting for Clamp Cylinder A1 Return... Check Q1.1...' | German: 'S1_Prompts German 421' | French: 'S1_Prompts French 421'
  422 = 'Spare' | German: 'S1_Prompts German 422' | French: 'S1_Prompts French 422'
  423 = 'Spare' | German: 'S1_Prompts German 423' | French: 'S1_Prompts French 423'
  424 = 'Spare' | German: 'S1_Prompts German 424' | French: 'S1_Prompts French 424'
  425 = 'Spare' | German: 'S1_Prompts German 425' | French: 'S1_Prompts French 425'
  426 = 'Spare' | German: 'S1_Prompts German 426' | French: 'S1_Prompts French 426'
  427 = 'Spare' | German: 'S1_Prompts German 427' | French: 'S1_Prompts French 427'
  428 = 'Spare' | German: 'S1_Prompts German 428' | French: 'S1_Prompts French 428'
  429 = 'Spare' | German: 'S1_Prompts German 429' | French: 'S1_Prompts French 429'
  430 = 'Waiting for Clamp Cylinder A1 Advance... Check Q1.0...' | German: 'S1_Prompts German 430' | French: 'S1_Prompts French 430'
  431 = 'Waiting for Clamp Cylinder A1 Return... Check Q1.1...' | German: 'S1_Prompts German 431' | French: 'S1_Prompts French 431'
  432 = 'Spare' | German: 'S1_Prompts German 432' | French: 'S1_Prompts French 432'
  433 = 'Spare' | German: 'S1_Prompts German 433' | French: 'S1_Prompts French 433'
  434 = 'Spare' | German: 'S1_Prompts German 434' | French: 'S1_Prompts French 434'
  435 = 'Spare' | German: 'S1_Prompts German 435' | French: 'S1_Prompts French 435'
  436 = 'Spare' | German: 'S1_Prompts German 436' | French: 'S1_Prompts French 436'
  437 = 'Spare' | German: 'S1_Prompts German 437' | French: 'S1_Prompts French 437'
  438 = 'Spare' | German: 'S1_Prompts German 438' | French: 'S1_Prompts French 438'
  439 = 'Spare' | German: 'S1_Prompts German 439' | French: 'S1_Prompts French 439'
  440 = 'Waiting for Clamp Cylinder A1 Advance... Check Q1.0...' | German: 'S1_Prompts German 440' | French: 'S1_Prompts French 440'
  441 = 'Waiting for Clamp Cylinder A1 Return... Check Q1.1...' | German: 'S1_Prompts German 441' | French: 'S1_Prompts French 441'
  442 = 'Spare' | German: 'S1_Prompts German 442' | French: 'S1_Prompts French 442'
  443 = 'Spare' | German: 'S1_Prompts German 443' | French: 'S1_Prompts French 443'
  444 = 'Spare' | German: 'S1_Prompts German 444' | French: 'S1_Prompts French 444'
  445 = 'Spare' | German: 'S1_Prompts German 445' | French: 'S1_Prompts French 445'
  446 = 'Spare' | German: 'S1_Prompts German 446' | French: 'S1_Prompts French 446'
  447 = 'Spare' | German: 'S1_Prompts German 447' | French: 'S1_Prompts French 447'
  448 = 'Spare' | German: 'S1_Prompts German 448' | French: 'S1_Prompts French 448'
  449 = 'Spare' | German: 'S1_Prompts German 449' | French: 'S1_Prompts French 449'
  450 = 'Waiting for Clamp Cylinder A1 Advance... Check Q1.0...' | German: 'S1_Prompts German 450' | French: 'S1_Prompts French 450'
  451 = 'Waiting for Clamp Cylinder A1 Return... Check Q1.1...' | German: 'S1_Prompts German 451' | French: 'S1_Prompts French 451'
  452 = 'Spare' | German: 'S1_Prompts German 452' | French: 'S1_Prompts French 452'
  453 = 'Spare' | German: 'S1_Prompts German 453' | French: 'S1_Prompts French 453'
  454 = 'Spare' | German: 'S1_Prompts German 454' | French: 'S1_Prompts French 454'
  455 = 'Spare' | German: 'S1_Prompts German 455' | French: 'S1_Prompts French 455'
  456 = 'Spare' | German: 'S1_Prompts German 456' | French: 'S1_Prompts French 456'
  457 = 'Spare' | German: 'S1_Prompts German 457' | French: 'S1_Prompts French 457'
  458 = 'Spare' | German: 'S1_Prompts German 458' | French: 'S1_Prompts French 458'
  459 = 'Spare' | German: 'S1_Prompts German 459' | French: 'S1_Prompts French 459'
  460 = 'Waiting for Clamp Cylinder A1 Advance... Check Q1.0...' | German: 'S1_Prompts German 460' | French: 'S1_Prompts French 460'
  461 = 'Waiting for Clamp Cylinder A1 Return... Check Q1.1...' | German: 'S1_Prompts German 461' | French: 'S1_Prompts French 461'
  462 = 'Spare' | German: 'S1_Prompts German 462' | French: 'S1_Prompts French 462'
  463 = 'Spare' | German: 'S1_Prompts German 463' | French: 'S1_Prompts French 463'
  464 = 'Spare' | German: 'S1_Prompts German 464' | French: 'S1_Prompts French 464'
  465 = 'Spare' | German: 'S1_Prompts German 465' | French: 'S1_Prompts French 465'
  466 = 'Spare' | German: 'S1_Prompts German 466' | French: 'S1_Prompts French 466'
  467 = 'Spare' | German: 'S1_Prompts German 467' | French: 'S1_Prompts French 467'
  468 = 'Spare' | German: 'S1_Prompts German 468' | French: 'S1_Prompts French 468'
  469 = 'Spare' | German: 'S1_Prompts German 469' | French: 'S1_Prompts French 469'
  470 = 'Waiting for Clamp Cylinder A1 Advance... Check Q1.0...' | German: 'S1_Prompts German 470' | French: 'S1_Prompts French 470'
  471 = 'Waiting for Clamp Cylinder A1 Return... Check Q1.1...' | German: 'S1_Prompts German 471' | French: 'S1_Prompts French 471'
  472 = 'Spare' | German: 'S1_Prompts German 472' | French: 'S1_Prompts French 472'
  473 = 'Spare' | German: 'S1_Prompts German 473' | French: 'S1_Prompts French 473'
  474 = 'Spare' | German: 'S1_Prompts German 474' | French: 'S1_Prompts French 474'
  475 = 'Spare' | German: 'S1_Prompts German 475' | French: 'S1_Prompts French 475'
  476 = 'Spare' | German: 'S1_Prompts German 476' | French: 'S1_Prompts French 476'
  477 = 'Spare' | German: 'S1_Prompts German 477' | French: 'S1_Prompts French 477'
  478 = 'Spare' | German: 'S1_Prompts German 478' | French: 'S1_Prompts French 478'
  479 = 'Spare' | German: 'S1_Prompts German 479' | French: 'S1_Prompts French 479'
  480 = 'Waiting for Clamp Cylinder A1 Advance... Check Q1.0...' | German: 'S1_Prompts German 480' | French: 'S1_Prompts French 480'
  481 = 'Waiting for Clamp Cylinder A1 Return... Check Q1.1...' | German: 'S1_Prompts German 481' | French: 'S1_Prompts French 481'
  482 = 'Spare' | German: 'S1_Prompts German 482' | French: 'S1_Prompts French 482'
  483 = 'Spare' | German: 'S1_Prompts German 483' | French: 'S1_Prompts French 483'
  484 = 'Spare' | German: 'S1_Prompts German 484' | French: 'S1_Prompts French 484'
  485 = 'Spare' | German: 'S1_Prompts German 485' | French: 'S1_Prompts French 485'
  486 = 'Spare' | German: 'S1_Prompts German 486' | French: 'S1_Prompts French 486'
  487 = 'Spare' | German: 'S1_Prompts German 487' | French: 'S1_Prompts French 487'
  488 = 'Spare' | German: 'S1_Prompts German 488' | French: 'S1_Prompts French 488'
  489 = 'Spare' | German: 'S1_Prompts German 489' | French: 'S1_Prompts French 489'
  490 = 'Waiting for Clamp Cylinder A1 Advance... Check Q1.0...' | German: 'S1_Prompts German 490' | French: 'S1_Prompts French 490'
  491 = 'Waiting for Clamp Cylinder A1 Return... Check Q1.1...' | German: 'S1_Prompts German 491' | French: 'S1_Prompts French 491'
  492 = 'Spare' | German: 'S1_Prompts German 492' | French: 'S1_Prompts French 492'
  493 = 'Spare' | German: 'S1_Prompts German 493' | French: 'S1_Prompts French 493'
  494 = 'Spare' | German: 'S1_Prompts German 494' | French: 'S1_Prompts French 494'
  495 = 'Spare' | German: 'S1_Prompts German 495' | French: 'S1_Prompts French 495'
  496 = 'Spare' | German: 'S1_Prompts German 496' | French: 'S1_Prompts French 496'
  497 = 'Spare' | German: 'S1_Prompts German 497' | French: 'S1_Prompts French 497'
  498 = 'Spare' | German: 'S1_Prompts German 498' | French: 'S1_Prompts French 498'
  499 = 'Spare' | German: 'S1_Prompts German 499' | French: 'S1_Prompts French 499'
  500 = 'Waiting for Clamp Cylinder A1 Advance... Check Q1.0...' | German: 'S1_Prompts German 500' | French: 'S1_Prompts French 500'
  501 = 'Waiting for Clamp Cylinder A1 Return... Check Q1.1...' | German: 'S1_Prompts German 501' | French: 'S1_Prompts French 501'
  502 = 'Spare' | German: 'S1_Prompts German 502' | French: 'S1_Prompts French 502'
  503 = 'Spare' | German: 'S1_Prompts German 503' | French: 'S1_Prompts French 503'
  504 = 'Spare' | German: 'S1_Prompts German 504' | French: 'S1_Prompts French 504'
  505 = 'Spare' | German: 'S1_Prompts German 505' | French: 'S1_Prompts French 505'
  506 = 'Spare' | German: 'S1_Prompts German 506' | French: 'S1_Prompts French 506'
  507 = 'Spare' | German: 'S1_Prompts German 507' | French: 'S1_Prompts French 507'
  508 = 'Spare' | German: 'S1_Prompts German 508' | French: 'S1_Prompts French 508'
  509 = 'Spare' | German: 'S1_Prompts German 509' | French: 'S1_Prompts French 509'
  510 = 'Waiting for Clamp Cylinder A1 Advance... Check Q1.0...' | German: 'S1_Prompts German 510' | French: 'S1_Prompts French 510'
  511 = 'Waiting for Clamp Cylinder A1 Return... Check Q1.1...' | German: 'S1_Prompts German 511' | French: 'S1_Prompts French 511'
  512 = 'Spare' | German: 'S1_Prompts German 512' | French: 'S1_Prompts French 512'
  513 = 'Spare' | German: 'S1_Prompts German 513' | French: 'S1_Prompts French 513'
  514 = 'Spare' | German: 'S1_Prompts German 514' | French: 'S1_Prompts French 514'
  515 = 'Spare' | German: 'S1_Prompts German 515' | French: 'S1_Prompts French 515'
  516 = 'Spare' | German: 'S1_Prompts German 516' | French: 'S1_Prompts French 516'
  517 = 'Spare' | German: 'S1_Prompts German 517' | French: 'S1_Prompts French 517'
  518 = 'Spare' | German: 'S1_Prompts German 518' | French: 'S1_Prompts French 518'
  519 = 'Spare' | German: 'S1_Prompts German 519' | French: 'S1_Prompts French 519'
  520 = 'Waiting for Clamp Cylinder A1 Advance... Check Q1.0...' | German: 'S1_Prompts German 520' | French: 'S1_Prompts French 520'
  521 = 'Waiting for Clamp Cylinder A1 Return... Check Q1.1...' | German: 'S1_Prompts German 521' | French: 'S1_Prompts French 521'
  522 = 'Spare' | German: 'S1_Prompts German 522' | French: 'S1_Prompts French 522'
  523 = 'Spare' | German: 'S1_Prompts German 523' | French: 'S1_Prompts French 523'
  524 = 'Spare' | German: 'S1_Prompts German 524' | French: 'S1_Prompts French 524'
  525 = 'Spare' | German: 'S1_Prompts German 525' | French: 'S1_Prompts French 525'
  526 = 'Spare' | German: 'S1_Prompts German 526' | French: 'S1_Prompts French 526'
  527 = 'Spare' | German: 'S1_Prompts German 527' | French: 'S1_Prompts French 527'
  528 = 'Spare' | German: 'S1_Prompts German 528' | French: 'S1_Prompts French 528'
  529 = 'Spare' | German: 'S1_Prompts German 529' | French: 'S1_Prompts French 529'
  530 = 'Waiting for Clamp Cylinder A1 Advance... Check Q1.0...' | German: 'S1_Prompts German 530' | French: 'S1_Prompts French 530'
  531 = 'Waiting for Clamp Cylinder A1 Return... Check Q1.1...' | German: 'S1_Prompts German 531' | French: 'S1_Prompts French 531'
  532 = 'Spare' | German: 'S1_Prompts German 532' | French: 'S1_Prompts French 532'
  533 = 'Spare' | German: 'S1_Prompts German 533' | French: 'S1_Prompts French 533'
  534 = 'Spare' | German: 'S1_Prompts German 534' | French: 'S1_Prompts French 534'
  535 = 'Spare' | German: 'S1_Prompts German 535' | French: 'S1_Prompts French 535'
  536 = 'Spare' | German: 'S1_Prompts German 536' | French: 'S1_Prompts French 536'
  537 = 'Spare' | German: 'S1_Prompts German 537' | French: 'S1_Prompts French 537'
  538 = 'Spare' | German: 'S1_Prompts German 538' | French: 'S1_Prompts French 538'
  539 = 'Spare' | German: 'S1_Prompts German 539' | French: 'S1_Prompts French 539'
  540 = 'Waiting for Clamp Cylinder A1 Advance... Check Q1.0...' | German: 'S1_Prompts German 540' | French: 'S1_Prompts French 540'
  541 = 'Waiting for Clamp Cylinder A1 Return... Check Q1.1...' | German: 'S1_Prompts German 541' | French: 'S1_Prompts French 541'
  542 = 'Spare' | German: 'S1_Prompts German 542' | French: 'S1_Prompts French 542'
  543 = 'Spare' | German: 'S1_Prompts German 543' | French: 'S1_Prompts French 543'
  544 = 'Spare' | German: 'S1_Prompts German 544' | French: 'S1_Prompts French 544'
  545 = 'Spare' | German: 'S1_Prompts German 545' | French: 'S1_Prompts French 545'
  546 = 'Spare' | German: 'S1_Prompts German 546' | French: 'S1_Prompts French 546'
  547 = 'Spare' | German: 'S1_Prompts German 547' | French: 'S1_Prompts French 547'
  548 = 'Spare' | German: 'S1_Prompts German 548' | French: 'S1_Prompts French 548'
  549 = 'Spare' | German: 'S1_Prompts German 549' | French: 'S1_Prompts French 549'
  550 = 'Waiting for Clamp Cylinder A1 Advance... Check Q1.0...' | German: 'S1_Prompts German 550' | French: 'S1_Prompts French 550'
  551 = 'Waiting for Clamp Cylinder A1 Return... Check Q1.1...' | German: 'S1_Prompts German 551' | French: 'S1_Prompts French 551'
  552 = 'Spare' | German: 'S1_Prompts German 552' | French: 'S1_Prompts French 552'
  553 = 'Spare' | German: 'S1_Prompts German 553' | French: 'S1_Prompts French 553'
  554 = 'Spare' | German: 'S1_Prompts German 554' | French: 'S1_Prompts French 554'
  555 = 'Spare' | German: 'S1_Prompts German 555' | French: 'S1_Prompts French 555'
  556 = 'Spare' | German: 'S1_Prompts German 556' | French: 'S1_Prompts French 556'
  557 = 'Spare' | German: 'S1_Prompts German 557' | French: 'S1_Prompts French 557'
  558 = 'Spare' | German: 'S1_Prompts German 558' | French: 'S1_Prompts French 558'
  559 = 'Spare' | German: 'S1_Prompts German 559' | French: 'S1_Prompts French 559'
  560 = 'Waiting for Clamp Cylinder A1 Advance... Check Q1.0...' | German: 'S1_Prompts German 560' | French: 'S1_Prompts French 560'
  561 = 'Waiting for Clamp Cylinder A1 Return... Check Q1.1...' | German: 'S1_Prompts German 561' | French: 'S1_Prompts French 561'
  562 = 'Spare' | German: 'S1_Prompts German 562' | French: 'S1_Prompts French 562'
  563 = 'Spare' | German: 'S1_Prompts German 563' | French: 'S1_Prompts French 563'
  564 = 'Spare' | German: 'S1_Prompts German 564' | French: 'S1_Prompts French 564'
  565 = 'Spare' | German: 'S1_Prompts German 565' | French: 'S1_Prompts French 565'
  566 = 'Spare' | German: 'S1_Prompts German 566' | French: 'S1_Prompts French 566'
  567 = 'Spare' | German: 'S1_Prompts German 567' | French: 'S1_Prompts French 567'
  568 = 'Spare' | German: 'S1_Prompts German 568' | French: 'S1_Prompts French 568'
  569 = 'Spare' | German: 'S1_Prompts German 569' | French: 'S1_Prompts French 569'
  570 = 'Waiting for Clamp Cylinder A1 Advance... Check Q1.0...' | German: 'S1_Prompts German 570' | French: 'S1_Prompts French 570'
  571 = 'Waiting for Clamp Cylinder A1 Return... Check Q1.1...' | German: 'S1_Prompts German 571' | French: 'S1_Prompts French 571'
  572 = 'Spare' | German: 'S1_Prompts German 572' | French: 'S1_Prompts French 572'
  573 = 'Spare' | German: 'S1_Prompts German 573' | French: 'S1_Prompts French 573'
  574 = 'Spare' | German: 'S1_Prompts German 574' | French: 'S1_Prompts French 574'
  575 = 'Spare' | German: 'S1_Prompts German 575' | French: 'S1_Prompts French 575'
  576 = 'Spare' | German: 'S1_Prompts German 576' | French: 'S1_Prompts French 576'
  577 = 'Spare' | German: 'S1_Prompts German 577' | French: 'S1_Prompts French 577'
  578 = 'Spare' | German: 'S1_Prompts German 578' | French: 'S1_Prompts French 578'
  579 = 'Spare' | German: 'S1_Prompts German 579' | French: 'S1_Prompts French 579'
  580 = 'Waiting for Clamp Cylinder A1 Advance... Check Q1.0...' | German: 'S1_Prompts German 580' | French: 'S1_Prompts French 580'
  581 = 'Waiting for Clamp Cylinder A1 Return... Check Q1.1...' | German: 'S1_Prompts German 581' | French: 'S1_Prompts French 581'
  582 = 'Spare' | German: 'S1_Prompts German 582' | French: 'S1_Prompts French 582'
  583 = 'Spare' | German: 'S1_Prompts German 583' | French: 'S1_Prompts French 583'
  584 = 'Spare' | German: 'S1_Prompts German 584' | French: 'S1_Prompts French 584'
  585 = 'Spare' | German: 'S1_Prompts German 585' | French: 'S1_Prompts French 585'
  586 = 'Spare' | German: 'S1_Prompts German 586' | French: 'S1_Prompts French 586'
  587 = 'Spare' | German: 'S1_Prompts German 587' | French: 'S1_Prompts French 587'
  588 = 'Spare' | German: 'S1_Prompts German 588' | French: 'S1_Prompts French 588'
  589 = 'Spare' | German: 'S1_Prompts German 589' | French: 'S1_Prompts French 589'
  590 = 'Waiting for Clamp Cylinder A1 Advance... Check Q1.0...' | German: 'S1_Prompts German 590' | French: 'S1_Prompts French 590'
  591 = 'Waiting for Clamp Cylinder A1 Return... Check Q1.1...' | German: 'S1_Prompts German 591' | French: 'S1_Prompts French 591'
  592 = 'Spare' | German: 'S1_Prompts German 592' | French: 'S1_Prompts French 592'
  593 = 'Spare' | German: 'S1_Prompts German 593' | French: 'S1_Prompts French 593'
  594 = 'Spare' | German: 'S1_Prompts German 594' | French: 'S1_Prompts French 594'
  595 = 'Spare' | German: 'S1_Prompts German 595' | French: 'S1_Prompts French 595'
  596 = 'Spare' | German: 'S1_Prompts German 596' | French: 'S1_Prompts French 596'
  597 = 'Spare' | German: 'S1_Prompts German 597' | French: 'S1_Prompts French 597'
  598 = 'Spare' | German: 'S1_Prompts German 598' | French: 'S1_Prompts French 598'
  599 = 'Spare' | German: 'S1_Prompts German 599' | French: 'S1_Prompts French 599'
  600 = 'Waiting for Clamp Cylinder A1 Advance... Check Q1.0...' | German: 'S1_Prompts German 600' | French: 'S1_Prompts French 600'
  601 = 'Waiting for Clamp Cylinder A1 Return... Check Q1.1...' | German: 'S1_Prompts German 601' | French: 'S1_Prompts French 601'
  602 = 'Spare' | German: 'S1_Prompts German 602' | French: 'S1_Prompts French 602'
  603 = 'Spare' | German: 'S1_Prompts German 603' | French: 'S1_Prompts French 603'
  604 = 'Spare' | German: 'S1_Prompts German 604' | French: 'S1_Prompts French 604'
  605 = 'Spare' | German: 'S1_Prompts German 605' | French: 'S1_Prompts French 605'
  606 = 'Spare' | German: 'S1_Prompts German 606' | French: 'S1_Prompts French 606'
  607 = 'Spare' | German: 'S1_Prompts German 607' | French: 'S1_Prompts French 607'
  608 = 'Spare' | German: 'S1_Prompts German 608' | French: 'S1_Prompts French 608'
  609 = 'Spare' | German: 'S1_Prompts German 609' | French: 'S1_Prompts French 609'
  610 = 'Waiting for Clamp Cylinder A1 Advance... Check Q1.0...' | German: 'S1_Prompts German 610' | French: 'S1_Prompts French 610'
  611 = 'Waiting for Clamp Cylinder A1 Return... Check Q1.1...' | German: 'S1_Prompts German 611' | French: 'S1_Prompts French 611'
  612 = 'Spare' | German: 'S1_Prompts German 612' | French: 'S1_Prompts French 612'
  613 = 'Spare' | German: 'S1_Prompts German 613' | French: 'S1_Prompts French 613'
  614 = 'Spare' | German: 'S1_Prompts German 614' | French: 'S1_Prompts French 614'
  615 = 'Spare' | German: 'S1_Prompts German 615' | French: 'S1_Prompts French 615'
  616 = 'Spare' | German: 'S1_Prompts German 616' | French: 'S1_Prompts French 616'
  617 = 'Spare' | German: 'S1_Prompts German 617' | French: 'S1_Prompts French 617'
  618 = 'Spare' | German: 'S1_Prompts German 618' | French: 'S1_Prompts French 618'
  619 = 'Spare' | German: 'S1_Prompts German 619' | French: 'S1_Prompts French 619'
  620 = 'Waiting for Clamp Cylinder A1 Advance... Check Q1.0...' | German: 'S1_Prompts German 620' | French: 'S1_Prompts French 620'
  621 = 'Waiting for Clamp Cylinder A1 Return... Check Q1.1...' | German: 'S1_Prompts German 621' | French: 'S1_Prompts French 621'
  622 = 'Spare' | German: 'S1_Prompts German 622' | French: 'S1_Prompts French 622'
  623 = 'Spare' | German: 'S1_Prompts German 623' | French: 'S1_Prompts French 623'
  624 = 'Spare' | German: 'S1_Prompts German 624' | French: 'S1_Prompts French 624'
  625 = 'Spare' | German: 'S1_Prompts German 625' | French: 'S1_Prompts French 625'
  626 = 'Spare' | German: 'S1_Prompts German 626' | French: 'S1_Prompts French 626'
  627 = 'Spare' | German: 'S1_Prompts German 627' | French: 'S1_Prompts French 627'
  628 = 'Spare' | German: 'S1_Prompts German 628' | French: 'S1_Prompts French 628'
  629 = 'Spare' | German: 'S1_Prompts German 629' | French: 'S1_Prompts French 629'
  630 = 'Waiting for Clamp Cylinder A1 Advance... Check Q1.0...' | German: 'S1_Prompts German 630' | French: 'S1_Prompts French 630'
  631 = 'Waiting for Clamp Cylinder A1 Return... Check Q1.1...' | German: 'S1_Prompts German 631' | French: 'S1_Prompts French 631'
  632 = 'Spare' | German: 'S1_Prompts German 632' | French: 'S1_Prompts French 632'
  633 = 'Spare' | German: 'S1_Prompts German 633' | French: 'S1_Prompts French 633'
  634 = 'Spare' | German: 'S1_Prompts German 634' | French: 'S1_Prompts French 634'
  635 = 'Spare' | German: 'S1_Prompts German 635' | French: 'S1_Prompts French 635'
  636 = 'Spare' | German: 'S1_Prompts German 636' | French: 'S1_Prompts French 636'
  637 = 'Spare' | German: 'S1_Prompts German 637' | French: 'S1_Prompts French 637'
  638 = 'Spare' | German: 'S1_Prompts German 638' | French: 'S1_Prompts French 638'
  639 = 'Spare' | German: 'S1_Prompts German 639' | French: 'S1_Prompts French 639'
  640 = 'Waiting for Clamp Cylinder A1 Advance... Check Q1.0...' | German: 'S1_Prompts German 640' | French: 'S1_Prompts French 640'
  641 = 'Waiting for Clamp Cylinder A1 Return... Check Q1.1...' | German: 'S1_Prompts German 641' | French: 'S1_Prompts French 641'
  642 = 'Spare' | German: 'S1_Prompts German 642' | French: 'S1_Prompts French 642'
  643 = 'Spare' | German: 'S1_Prompts German 643' | French: 'S1_Prompts French 643'
  644 = 'Spare' | German: 'S1_Prompts German 644' | French: 'S1_Prompts French 644'
  645 = 'Spare' | German: 'S1_Prompts German 645' | French: 'S1_Prompts French 645'
  646 = 'Spare' | German: 'S1_Prompts German 646' | French: 'S1_Prompts French 646'
  647 = 'Spare' | German: 'S1_Prompts German 647' | French: 'S1_Prompts French 647'
  648 = 'Spare' | German: 'S1_Prompts German 648' | French: 'S1_Prompts French 648'
  649 = 'Spare' | German: 'S1_Prompts German 649' | French: 'S1_Prompts French 649'
  650 = 'Waiting for Clamp Cylinder A1 Advance... Check Q1.0...' | German: 'S1_Prompts German 650' | French: 'S1_Prompts French 650'
  651 = 'Waiting for Clamp Cylinder A1 Return... Check Q1.1...' | German: 'S1_Prompts German 651' | French: 'S1_Prompts French 651'
  652 = 'Spare' | German: 'S1_Prompts German 652' | French: 'S1_Prompts French 652'
  653 = 'Spare' | German: 'S1_Prompts German 653' | French: 'S1_Prompts French 653'
  654 = 'Spare' | German: 'S1_Prompts German 654' | French: 'S1_Prompts French 654'
  655 = 'Spare' | German: 'S1_Prompts German 655' | French: 'S1_Prompts French 655'
  656 = 'Spare' | German: 'S1_Prompts German 656' | French: 'S1_Prompts French 656'
  657 = 'Spare' | German: 'S1_Prompts German 657' | French: 'S1_Prompts French 657'
  658 = 'Spare' | German: 'S1_Prompts German 658' | French: 'S1_Prompts French 658'
  659 = 'Spare' | German: 'S1_Prompts German 659' | French: 'S1_Prompts French 659'
  660 = 'Waiting for Clamp Cylinder A1 Advance... Check Q1.0...' | German: 'S1_Prompts German 660' | French: 'S1_Prompts French 660'
  661 = 'Waiting for Clamp Cylinder A1 Return... Check Q1.1...' | German: 'S1_Prompts German 661' | French: 'S1_Prompts French 661'
  662 = 'Spare' | German: 'S1_Prompts German 662' | French: 'S1_Prompts French 662'
  663 = 'Spare' | German: 'S1_Prompts German 663' | French: 'S1_Prompts French 663'
  664 = 'Spare' | German: 'S1_Prompts German 664' | French: 'S1_Prompts French 664'
  665 = 'Spare' | German: 'S1_Prompts German 665' | French: 'S1_Prompts French 665'
  666 = 'Spare' | German: 'S1_Prompts German 666' | French: 'S1_Prompts French 666'
  667 = 'Spare' | German: 'S1_Prompts German 667' | French: 'S1_Prompts French 667'
  668 = 'Spare' | German: 'S1_Prompts German 668' | French: 'S1_Prompts French 668'
  669 = 'Spare' | German: 'S1_Prompts German 669' | French: 'S1_Prompts French 669'
  670 = 'Waiting for Clamp Cylinder A1 Advance... Check Q1.0...' | German: 'S1_Prompts German 670' | French: 'S1_Prompts French 670'
  671 = 'Waiting for Clamp Cylinder A1 Return... Check Q1.1...' | German: 'S1_Prompts German 671' | French: 'S1_Prompts French 671'
  672 = 'Spare' | German: 'S1_Prompts German 672' | French: 'S1_Prompts French 672'
  673 = 'Spare' | German: 'S1_Prompts German 673' | French: 'S1_Prompts French 673'
  674 = 'Spare' | German: 'S1_Prompts German 674' | French: 'S1_Prompts French 674'
  675 = 'Spare' | German: 'S1_Prompts German 675' | French: 'S1_Prompts French 675'
  676 = 'Spare' | German: 'S1_Prompts German 676' | French: 'S1_Prompts French 676'
  677 = 'Spare' | German: 'S1_Prompts German 677' | French: 'S1_Prompts French 677'
  678 = 'Spare' | German: 'S1_Prompts German 678' | French: 'S1_Prompts French 678'
  679 = 'Spare' | German: 'S1_Prompts German 679' | French: 'S1_Prompts French 679'
  680 = 'Waiting for Clamp Cylinder A1 Advance... Check Q1.0...' | German: 'S1_Prompts German 680' | French: 'S1_Prompts French 680'
  681 = 'Waiting for Clamp Cylinder A1 Return... Check Q1.1...' | German: 'S1_Prompts German 681' | French: 'S1_Prompts French 681'
  682 = 'Spare' | German: 'S1_Prompts German 682' | French: 'S1_Prompts French 682'
  683 = 'Spare' | German: 'S1_Prompts German 683' | French: 'S1_Prompts French 683'
  684 = 'Spare' | German: 'S1_Prompts German 684' | French: 'S1_Prompts French 684'
  685 = 'Spare' | German: 'S1_Prompts German 685' | French: 'S1_Prompts French 685'
  686 = 'Spare' | German: 'S1_Prompts German 686' | French: 'S1_Prompts French 686'
  687 = 'Spare' | German: 'S1_Prompts German 687' | French: 'S1_Prompts French 687'
  688 = 'Spare' | German: 'S1_Prompts German 688' | French: 'S1_Prompts French 688'
  689 = 'Spare' | German: 'S1_Prompts German 689' | French: 'S1_Prompts French 689'
  690 = 'Waiting for Clamp Cylinder A1 Advance... Check Q1.0...' | German: 'S1_Prompts German 690' | French: 'S1_Prompts French 690'
  691 = 'Waiting for Clamp Cylinder A1 Return... Check Q1.1...' | German: 'S1_Prompts German 691' | French: 'S1_Prompts French 691'
  692 = 'Spare' | German: 'S1_Prompts German 692' | French: 'S1_Prompts French 692'
  693 = 'Spare' | German: 'S1_Prompts German 693' | French: 'S1_Prompts French 693'
  694 = 'Spare' | German: 'S1_Prompts German 694' | French: 'S1_Prompts French 694'
  695 = 'Spare' | German: 'S1_Prompts German 695' | French: 'S1_Prompts French 695'
  696 = 'Spare' | German: 'S1_Prompts German 696' | French: 'S1_Prompts French 696'
  697 = 'Spare' | German: 'S1_Prompts German 697' | French: 'S1_Prompts French 697'
  698 = 'Spare' | German: 'S1_Prompts German 698' | French: 'S1_Prompts French 698'
  699 = 'Spare' | German: 'S1_Prompts German 699' | French: 'S1_Prompts French 699'
  700 = 'Waiting for Clamp Cylinder A1 Advance... Check Q1.0...' | German: 'S1_Prompts German 700' | French: 'S1_Prompts French 700'
  701 = 'Waiting for Clamp Cylinder A1 Return... Check Q1.1...' | German: 'S1_Prompts German 701' | French: 'S1_Prompts French 701'
  702 = 'Spare' | German: 'S1_Prompts German 702' | French: 'S1_Prompts French 702'
  703 = 'Spare' | German: 'S1_Prompts German 703' | French: 'S1_Prompts French 703'
  704 = 'Spare' | German: 'S1_Prompts German 704' | French: 'S1_Prompts French 704'
  705 = 'Spare' | German: 'S1_Prompts German 705' | French: 'S1_Prompts French 705'
  706 = 'Spare' | German: 'S1_Prompts German 706' | French: 'S1_Prompts French 706'
  707 = 'Spare' | German: 'S1_Prompts German 707' | French: 'S1_Prompts French 707'
  708 = 'Spare' | German: 'S1_Prompts German 708' | French: 'S1_Prompts French 708'
  709 = 'Spare' | German: 'S1_Prompts German 709' | French: 'S1_Prompts French 709'
  710 = 'Waiting for Clamp Cylinder A1 Advance... Check Q1.0...' | German: 'S1_Prompts German 710' | French: 'S1_Prompts French 710'
  711 = 'Waiting for Clamp Cylinder A1 Return... Check Q1.1...' | German: 'S1_Prompts German 711' | French: 'S1_Prompts French 711'
  712 = 'Spare' | German: 'S1_Prompts German 712' | French: 'S1_Prompts French 712'
  713 = 'Spare' | German: 'S1_Prompts German 713' | French: 'S1_Prompts French 713'
  714 = 'Spare' | German: 'S1_Prompts German 714' | French: 'S1_Prompts French 714'
  715 = 'Spare' | German: 'S1_Prompts German 715' | French: 'S1_Prompts French 715'
  716 = 'Spare' | German: 'S1_Prompts German 716' | French: 'S1_Prompts French 716'
  717 = 'Spare' | German: 'S1_Prompts German 717' | French: 'S1_Prompts French 717'
  718 = 'Spare' | German: 'S1_Prompts German 718' | French: 'S1_Prompts French 718'
  719 = 'Spare' | German: 'S1_Prompts German 719' | French: 'S1_Prompts French 719'
  720 = 'Waiting for Clamp Cylinder A1 Advance... Check Q1.0...' | German: 'S1_Prompts German 720' | French: 'S1_Prompts French 720'
  721 = 'Waiting for Clamp Cylinder A1 Return... Check Q1.1...' | German: 'S1_Prompts German 721' | French: 'S1_Prompts French 721'
  722 = 'Spare' | German: 'S1_Prompts German 722' | French: 'S1_Prompts French 722'
  723 = 'Spare' | German: 'S1_Prompts German 723' | French: 'S1_Prompts French 723'
  724 = 'Spare' | German: 'S1_Prompts German 724' | French: 'S1_Prompts French 724'
  725 = 'Spare' | German: 'S1_Prompts German 725' | French: 'S1_Prompts French 725'
  726 = 'Spare' | German: 'S1_Prompts German 726' | French: 'S1_Prompts French 726'
  727 = 'Spare' | German: 'S1_Prompts German 727' | French: 'S1_Prompts French 727'
  728 = 'Spare' | German: 'S1_Prompts German 728' | French: 'S1_Prompts French 728'
  729 = 'Spare' | German: 'S1_Prompts German 729' | French: 'S1_Prompts French 729'
  730 = 'Waiting for Clamp Cylinder A1 Advance... Check Q1.0...' | German: 'S1_Prompts German 730' | French: 'S1_Prompts French 730'
  731 = 'Waiting for Clamp Cylinder A1 Return... Check Q1.1...' | German: 'S1_Prompts German 731' | French: 'S1_Prompts French 731'
  732 = 'Spare' | German: 'S1_Prompts German 732' | French: 'S1_Prompts French 732'
  733 = 'Spare' | German: 'S1_Prompts German 733' | French: 'S1_Prompts French 733'
  734 = 'Spare' | German: 'S1_Prompts German 734' | French: 'S1_Prompts French 734'
  735 = 'Spare' | German: 'S1_Prompts German 735' | French: 'S1_Prompts French 735'
  736 = 'Spare' | German: 'S1_Prompts German 736' | French: 'S1_Prompts French 736'
  737 = 'Spare' | German: 'S1_Prompts German 737' | French: 'S1_Prompts French 737'
  738 = 'Spare' | German: 'S1_Prompts German 738' | French: 'S1_Prompts French 738'
  739 = 'Spare' | German: 'S1_Prompts German 739' | French: 'S1_Prompts French 739'
  740 = 'Waiting for Clamp Cylinder A1 Advance... Check Q1.0...' | German: 'S1_Prompts German 740' | French: 'S1_Prompts French 740'
  741 = 'Waiting for Clamp Cylinder A1 Return... Check Q1.1...' | German: 'S1_Prompts German 741' | French: 'S1_Prompts French 741'
  742 = 'Spare' | German: 'S1_Prompts German 742' | French: 'S1_Prompts French 742'
  743 = 'Spare' | German: 'S1_Prompts German 743' | French: 'S1_Prompts French 743'
  744 = 'Spare' | German: 'S1_Prompts German 744' | French: 'S1_Prompts French 744'
  745 = 'Spare' | German: 'S1_Prompts German 745' | French: 'S1_Prompts French 745'
  746 = 'Spare' | German: 'S1_Prompts German 746' | French: 'S1_Prompts French 746'
  747 = 'Spare' | German: 'S1_Prompts German 747' | French: 'S1_Prompts French 747'
  748 = 'Spare' | German: 'S1_Prompts German 748' | French: 'S1_Prompts French 748'
  749 = 'Spare' | German: 'S1_Prompts German 749' | French: 'S1_Prompts French 749'
  750 = 'Waiting for Clamp Cylinder A1 Advance... Check Q1.0...' | German: 'S1_Prompts German 750' | French: 'S1_Prompts French 750'
  751 = 'Waiting for Clamp Cylinder A1 Return... Check Q1.1...' | German: 'S1_Prompts German 751' | French: 'S1_Prompts French 751'
  752 = 'Spare' | German: 'S1_Prompts German 752' | French: 'S1_Prompts French 752'
  753 = 'Spare' | German: 'S1_Prompts German 753' | French: 'S1_Prompts French 753'
  754 = 'Spare' | German: 'S1_Prompts German 754' | French: 'S1_Prompts French 754'
  755 = 'Spare' | German: 'S1_Prompts German 755' | French: 'S1_Prompts French 755'
  756 = 'Spare' | German: 'S1_Prompts German 756' | French: 'S1_Prompts French 756'
  757 = 'Spare' | German: 'S1_Prompts German 757' | French: 'S1_Prompts French 757'
  758 = 'Spare' | German: 'S1_Prompts German 758' | French: 'S1_Prompts French 758'
  759 = 'Spare' | German: 'S1_Prompts German 759' | French: 'S1_Prompts French 759'
  760 = 'Waiting for Clamp Cylinder A1 Advance... Check Q1.0...' | German: 'S1_Prompts German 760' | French: 'S1_Prompts French 760'
  761 = 'Waiting for Clamp Cylinder A1 Return... Check Q1.1...' | German: 'S1_Prompts German 761' | French: 'S1_Prompts French 761'
  762 = 'Spare' | German: 'S1_Prompts German 762' | French: 'S1_Prompts French 762'
  763 = 'Spare' | German: 'S1_Prompts German 763' | French: 'S1_Prompts French 763'
  764 = 'Spare' | German: 'S1_Prompts German 764' | French: 'S1_Prompts French 764'
  765 = 'Spare' | German: 'S1_Prompts German 765' | French: 'S1_Prompts French 765'
  766 = 'Spare' | German: 'S1_Prompts German 766' | French: 'S1_Prompts French 766'
  767 = 'Spare' | German: 'S1_Prompts German 767' | French: 'S1_Prompts French 767'
  768 = 'Spare' | German: 'S1_Prompts German 768' | French: 'S1_Prompts French 768'
  769 = 'Spare' | German: 'S1_Prompts German 769' | French: 'S1_Prompts French 769'
  770 = 'Waiting for Clamp Cylinder A1 Advance... Check Q1.0...' | German: 'S1_Prompts German 770' | French: 'S1_Prompts French 770'
  771 = 'Waiting for Clamp Cylinder A1 Return... Check Q1.1...' | German: 'S1_Prompts German 771' | French: 'S1_Prompts French 771'
  772 = 'Spare' | German: 'S1_Prompts German 772' | French: 'S1_Prompts French 772'
  773 = 'Spare' | German: 'S1_Prompts German 773' | French: 'S1_Prompts French 773'
  774 = 'Spare' | German: 'S1_Prompts German 774' | French: 'S1_Prompts French 774'
  775 = 'Spare' | German: 'S1_Prompts German 775' | French: 'S1_Prompts French 775'
  776 = 'Spare' | German: 'S1_Prompts German 776' | French: 'S1_Prompts French 776'
  777 = 'Spare' | German: 'S1_Prompts German 777' | French: 'S1_Prompts French 777'
  778 = 'Spare' | German: 'S1_Prompts German 778' | French: 'S1_Prompts French 778'
  779 = 'Spare' | German: 'S1_Prompts German 779' | French: 'S1_Prompts French 779'
  780 = 'Waiting for Clamp Cylinder A1 Advance... Check Q1.0...' | German: 'S1_Prompts German 780' | French: 'S1_Prompts French 780'
  781 = 'Waiting for Clamp Cylinder A1 Return... Check Q1.1...' | German: 'S1_Prompts German 781' | French: 'S1_Prompts French 781'
  782 = 'Spare' | German: 'S1_Prompts German 782' | French: 'S1_Prompts French 782'
  783 = 'Spare' | German: 'S1_Prompts German 783' | French: 'S1_Prompts French 783'
  784 = 'Spare' | German: 'S1_Prompts German 784' | French: 'S1_Prompts French 784'
  785 = 'Spare' | German: 'S1_Prompts German 785' | French: 'S1_Prompts French 785'
  786 = 'Spare' | German: 'S1_Prompts German 786' | French: 'S1_Prompts French 786'
  787 = 'Spare' | German: 'S1_Prompts German 787' | French: 'S1_Prompts French 787'
  788 = 'Spare' | German: 'S1_Prompts German 788' | French: 'S1_Prompts French 788'
  789 = 'Spare' | German: 'S1_Prompts German 789' | French: 'S1_Prompts French 789'
  790 = 'Waiting for Clamp Cylinder A1 Advance... Check Q1.0...' | German: 'S1_Prompts German 790' | French: 'S1_Prompts French 790'
  791 = 'Waiting for Clamp Cylinder A1 Return... Check Q1.1...' | German: 'S1_Prompts German 791' | French: 'S1_Prompts French 791'
  792 = 'Spare' | German: 'S1_Prompts German 792' | French: 'S1_Prompts French 792'
  793 = 'Spare' | German: 'S1_Prompts German 793' | French: 'S1_Prompts French 793'
  794 = 'Spare' | German: 'S1_Prompts German 794' | French: 'S1_Prompts French 794'
  795 = 'Spare' | German: 'S1_Prompts German 795' | French: 'S1_Prompts French 795'
  796 = 'Spare' | German: 'S1_Prompts German 796' | French: 'S1_Prompts French 796'
  797 = 'Spare' | German: 'S1_Prompts German 797' | French: 'S1_Prompts French 797'
  798 = 'Spare' | German: 'S1_Prompts German 798' | French: 'S1_Prompts French 798'
  799 = 'Spare' | German: 'S1_Prompts German 799' | French: 'S1_Prompts French 799'
  800 = 'Waiting for Clamp Cylinder A1 Advance... Check Q1.0...' | German: 'S1_Prompts German 800' | French: 'S1_Prompts French 800'
  801 = 'Waiting for Clamp Cylinder A1 Return... Check Q1.1...' | German: 'S1_Prompts German 801' | French: 'S1_Prompts French 801'
  802 = 'Spare' | German: 'S1_Prompts German 802' | French: 'S1_Prompts French 802'
  803 = 'Spare' | German: 'S1_Prompts German 803' | French: 'S1_Prompts French 803'
  804 = 'Spare' | German: 'S1_Prompts German 804' | French: 'S1_Prompts French 804'
  805 = 'Spare' | German: 'S1_Prompts German 805' | French: 'S1_Prompts French 805'
  806 = 'Spare' | German: 'S1_Prompts German 806' | French: 'S1_Prompts French 806'
  807 = 'Spare' | German: 'S1_Prompts German 807' | French: 'S1_Prompts French 807'
  808 = 'Spare' | German: 'S1_Prompts German 808' | French: 'S1_Prompts French 808'
  809 = 'Spare' | German: 'S1_Prompts German 809' | French: 'S1_Prompts French 809'
  810 = 'Waiting for Clamp Cylinder A1 Advance... Check Q1.0...' | German: 'S1_Prompts German 810' | French: 'S1_Prompts French 810'
  811 = 'Waiting for Clamp Cylinder A1 Return... Check Q1.1...' | German: 'S1_Prompts German 811' | French: 'S1_Prompts French 811'
  812 = 'Spare' | German: 'S1_Prompts German 812' | French: 'S1_Prompts French 812'
  813 = 'Spare' | German: 'S1_Prompts German 813' | French: 'S1_Prompts French 813'
  814 = 'Spare' | German: 'S1_Prompts German 814' | French: 'S1_Prompts French 814'
  815 = 'Spare' | German: 'S1_Prompts German 815' | French: 'S1_Prompts French 815'
  816 = 'Spare' | German: 'S1_Prompts German 816' | French: 'S1_Prompts French 816'
  817 = 'Spare' | German: 'S1_Prompts German 817' | French: 'S1_Prompts French 817'
  818 = 'Spare' | German: 'S1_Prompts German 818' | French: 'S1_Prompts French 818'
  819 = 'Spare' | German: 'S1_Prompts German 819' | French: 'S1_Prompts French 819'
  820 = 'Waiting for Clamp Cylinder A1 Advance... Check Q1.0...' | German: 'S1_Prompts German 820' | French: 'S1_Prompts French 820'
  821 = 'Waiting for Clamp Cylinder A1 Return... Check Q1.1...' | German: 'S1_Prompts German 821' | French: 'S1_Prompts French 821'
  822 = 'Spare' | German: 'S1_Prompts German 822' | French: 'S1_Prompts French 822'
  823 = 'Spare' | German: 'S1_Prompts German 823' | French: 'S1_Prompts French 823'
  824 = 'Spare' | German: 'S1_Prompts German 824' | French: 'S1_Prompts French 824'
  825 = 'Spare' | German: 'S1_Prompts German 825' | French: 'S1_Prompts French 825'
  826 = 'Spare' | German: 'S1_Prompts German 826' | French: 'S1_Prompts French 826'
  827 = 'Spare' | German: 'S1_Prompts German 827' | French: 'S1_Prompts French 827'
  828 = 'Spare' | German: 'S1_Prompts German 828' | French: 'S1_Prompts French 828'
  829 = 'Spare' | German: 'S1_Prompts German 829' | French: 'S1_Prompts French 829'
  830 = 'Waiting for Clamp Cylinder A1 Advance... Check Q1.0...' | German: 'S1_Prompts German 830' | French: 'S1_Prompts French 830'
  831 = 'Waiting for Clamp Cylinder A1 Return... Check Q1.1...' | German: 'S1_Prompts German 831' | French: 'S1_Prompts French 831'
  832 = 'Spare' | German: 'S1_Prompts German 832' | French: 'S1_Prompts French 832'
  833 = 'Spare' | German: 'S1_Prompts German 833' | French: 'S1_Prompts French 833'
  834 = 'Spare' | German: 'S1_Prompts German 834' | French: 'S1_Prompts French 834'
  835 = 'Spare' | German: 'S1_Prompts German 835' | French: 'S1_Prompts French 835'
  836 = 'Spare' | German: 'S1_Prompts German 836' | French: 'S1_Prompts French 836'
  837 = 'Spare' | German: 'S1_Prompts German 837' | French: 'S1_Prompts French 837'
  838 = 'Spare' | German: 'S1_Prompts German 838' | French: 'S1_Prompts French 838'
  839 = 'Spare' | German: 'S1_Prompts German 839' | French: 'S1_Prompts French 839'
  840 = 'Waiting for Clamp Cylinder A1 Advance... Check Q1.0...' | German: 'S1_Prompts German 840' | French: 'S1_Prompts French 840'
  841 = 'Waiting for Clamp Cylinder A1 Return... Check Q1.1...' | German: 'S1_Prompts German 841' | French: 'S1_Prompts French 841'
  842 = 'Spare' | German: 'S1_Prompts German 842' | French: 'S1_Prompts French 842'
  843 = 'Spare' | German: 'S1_Prompts German 843' | French: 'S1_Prompts French 843'
  844 = 'Spare' | German: 'S1_Prompts German 844' | French: 'S1_Prompts French 844'
  845 = 'Spare' | German: 'S1_Prompts German 845' | French: 'S1_Prompts French 845'
  846 = 'Spare' | German: 'S1_Prompts German 846' | French: 'S1_Prompts French 846'
  847 = 'Spare' | German: 'S1_Prompts German 847' | French: 'S1_Prompts French 847'
  848 = 'Spare' | German: 'S1_Prompts German 848' | French: 'S1_Prompts French 848'
  849 = 'Spare' | German: 'S1_Prompts German 849' | French: 'S1_Prompts French 849'
  850 = 'Waiting for Clamp Cylinder A1 Advance... Check Q1.0...' | German: 'S1_Prompts German 850' | French: 'S1_Prompts French 850'
  851 = 'Waiting for Clamp Cylinder A1 Return... Check Q1.1...' | German: 'S1_Prompts German 851' | French: 'S1_Prompts French 851'
  852 = 'Spare' | German: 'S1_Prompts German 852' | French: 'S1_Prompts French 852'
  853 = 'Spare' | German: 'S1_Prompts German 853' | French: 'S1_Prompts French 853'
  854 = 'Spare' | German: 'S1_Prompts German 854' | French: 'S1_Prompts French 854'
  855 = 'Spare' | German: 'S1_Prompts German 855' | French: 'S1_Prompts French 855'
  856 = 'Spare' | German: 'S1_Prompts German 856' | French: 'S1_Prompts French 856'
  857 = 'Spare' | German: 'S1_Prompts German 857' | French: 'S1_Prompts French 857'
  858 = 'Spare' | German: 'S1_Prompts German 858' | French: 'S1_Prompts French 858'
  859 = 'Spare' | German: 'S1_Prompts German 859' | French: 'S1_Prompts French 859'
  860 = 'Waiting for Clamp Cylinder A1 Advance... Check Q1.0...' | German: 'S1_Prompts German 860' | French: 'S1_Prompts French 860'
  861 = 'Waiting for Clamp Cylinder A1 Return... Check Q1.1...' | German: 'S1_Prompts German 861' | French: 'S1_Prompts French 861'
  862 = 'Spare' | German: 'S1_Prompts German 862' | French: 'S1_Prompts French 862'
  863 = 'Spare' | German: 'S1_Prompts German 863' | French: 'S1_Prompts French 863'
  864 = 'Spare' | German: 'S1_Prompts German 864' | French: 'S1_Prompts French 864'
  865 = 'Spare' | German: 'S1_Prompts German 865' | French: 'S1_Prompts French 865'
  866 = 'Spare' | German: 'S1_Prompts German 866' | French: 'S1_Prompts French 866'
  867 = 'Spare' | German: 'S1_Prompts German 867' | French: 'S1_Prompts French 867'
  868 = 'Spare' | German: 'S1_Prompts German 868' | French: 'S1_Prompts French 868'
  869 = 'Spare' | German: 'S1_Prompts German 869' | French: 'S1_Prompts French 869'
  870 = 'Waiting for Clamp Cylinder A1 Advance... Check Q1.0...' | German: 'S1_Prompts German 870' | French: 'S1_Prompts French 870'
  871 = 'Waiting for Clamp Cylinder A1 Return... Check Q1.1...' | German: 'S1_Prompts German 871' | French: 'S1_Prompts French 871'
  872 = 'Spare' | German: 'S1_Prompts German 872' | French: 'S1_Prompts French 872'
  873 = 'Spare' | German: 'S1_Prompts German 873' | French: 'S1_Prompts French 873'
  874 = 'Spare' | German: 'S1_Prompts German 874' | French: 'S1_Prompts French 874'
  875 = 'Spare' | German: 'S1_Prompts German 875' | French: 'S1_Prompts French 875'
  876 = 'Spare' | German: 'S1_Prompts German 876' | French: 'S1_Prompts French 876'
  877 = 'Spare' | German: 'S1_Prompts German 877' | French: 'S1_Prompts French 877'
  878 = 'Spare' | German: 'S1_Prompts German 878' | French: 'S1_Prompts French 878'
  879 = 'Spare' | German: 'S1_Prompts German 879' | French: 'S1_Prompts French 879'
  880 = 'Waiting for Clamp Cylinder A1 Advance... Check Q1.0...' | German: 'S1_Prompts German 880' | French: 'S1_Prompts French 880'
  881 = 'Waiting for Clamp Cylinder A1 Return... Check Q1.1...' | German: 'S1_Prompts German 881' | French: 'S1_Prompts French 881'
  882 = 'Spare' | German: 'S1_Prompts German 882' | French: 'S1_Prompts French 882'
  883 = 'Spare' | German: 'S1_Prompts German 883' | French: 'S1_Prompts French 883'
  884 = 'Spare' | German: 'S1_Prompts German 884' | French: 'S1_Prompts French 884'
  885 = 'Spare' | German: 'S1_Prompts German 885' | French: 'S1_Prompts French 885'
  886 = 'Spare' | German: 'S1_Prompts German 886' | French: 'S1_Prompts French 886'
  887 = 'Spare' | German: 'S1_Prompts German 887' | French: 'S1_Prompts French 887'
  888 = 'Spare' | German: 'S1_Prompts German 888' | French: 'S1_Prompts French 888'
  889 = 'Spare' | German: 'S1_Prompts German 889' | French: 'S1_Prompts French 889'
  890 = 'Waiting for Clamp Cylinder A1 Advance... Check Q1.0...' | German: 'S1_Prompts German 890' | French: 'S1_Prompts French 890'
  891 = 'Waiting for Clamp Cylinder A1 Return... Check Q1.1...' | German: 'S1_Prompts German 891' | French: 'S1_Prompts French 891'
  892 = 'Spare' | German: 'S1_Prompts German 892' | French: 'S1_Prompts French 892'
  893 = 'Spare' | German: 'S1_Prompts German 893' | French: 'S1_Prompts French 893'
  894 = 'Spare' | German: 'S1_Prompts German 894' | French: 'S1_Prompts French 894'
  895 = 'Spare' | German: 'S1_Prompts German 895' | French: 'S1_Prompts French 895'
  896 = 'Spare' | German: 'S1_Prompts German 896' | French: 'S1_Prompts French 896'
  897 = 'Spare' | German: 'S1_Prompts German 897' | French: 'S1_Prompts French 897'
  898 = 'Spare' | German: 'S1_Prompts German 898' | French: 'S1_Prompts French 898'
  899 = 'Spare' | German: 'S1_Prompts German 899' | French: 'S1_Prompts French 899'
  900 = 'Waiting for Clamp Cylinder A1 Advance... Check Q1.0...' | German: 'S1_Prompts German 900' | French: 'S1_Prompts French 900'
  901 = 'Waiting for Clamp Cylinder A1 Return... Check Q1.1...' | German: 'S1_Prompts German 901' | French: 'S1_Prompts French 901'
  902 = 'Spare' | German: 'S1_Prompts German 902' | French: 'S1_Prompts French 902'
  903 = 'Spare' | German: 'S1_Prompts German 903' | French: 'S1_Prompts French 903'
  904 = 'Spare' | German: 'S1_Prompts German 904' | French: 'S1_Prompts French 904'
  905 = 'Spare' | German: 'S1_Prompts German 905' | French: 'S1_Prompts French 905'
  906 = 'Spare' | German: 'S1_Prompts German 906' | French: 'S1_Prompts French 906'
  907 = 'Spare' | German: 'S1_Prompts German 907' | French: 'S1_Prompts French 907'
  908 = 'Spare' | German: 'S1_Prompts German 908' | French: 'S1_Prompts French 908'
  909 = 'Spare' | German: 'S1_Prompts German 909' | French: 'S1_Prompts French 909'
  910 = 'Waiting for Clamp Cylinder A1 Advance... Check Q1.0...' | German: 'S1_Prompts German 910' | French: 'S1_Prompts French 910'
  911 = 'Waiting for Clamp Cylinder A1 Return... Check Q1.1...' | German: 'S1_Prompts German 911' | French: 'S1_Prompts French 911'
  912 = 'Spare' | German: 'S1_Prompts German 912' | French: 'S1_Prompts French 912'
  913 = 'Spare' | German: 'S1_Prompts German 913' | French: 'S1_Prompts French 913'
  914 = 'Spare' | German: 'S1_Prompts German 914' | French: 'S1_Prompts French 914'
  915 = 'Spare' | German: 'S1_Prompts German 915' | French: 'S1_Prompts French 915'
  916 = 'Spare' | German: 'S1_Prompts German 916' | French: 'S1_Prompts French 916'
  917 = 'Spare' | German: 'S1_Prompts German 917' | French: 'S1_Prompts French 917'
  918 = 'Spare' | German: 'S1_Prompts German 918' | French: 'S1_Prompts French 918'
  919 = 'Spare' | German: 'S1_Prompts German 919' | French: 'S1_Prompts French 919'
  920 = 'Waiting for Clamp Cylinder A1 Advance... Check Q1.0...' | German: 'S1_Prompts German 920' | French: 'S1_Prompts French 920'
  921 = 'Waiting for Clamp Cylinder A1 Return... Check Q1.1...' | German: 'S1_Prompts German 921' | French: 'S1_Prompts French 921'
  922 = 'Spare' | German: 'S1_Prompts German 922' | French: 'S1_Prompts French 922'
  923 = 'Spare' | German: 'S1_Prompts German 923' | French: 'S1_Prompts French 923'
  924 = 'Spare' | German: 'S1_Prompts German 924' | French: 'S1_Prompts French 924'
  925 = 'Spare' | German: 'S1_Prompts German 925' | French: 'S1_Prompts French 925'
  926 = 'Spare' | German: 'S1_Prompts German 926' | French: 'S1_Prompts French 926'
  927 = 'Spare' | German: 'S1_Prompts German 927' | French: 'S1_Prompts French 927'
  928 = 'Spare' | German: 'S1_Prompts German 928' | French: 'S1_Prompts French 928'
  929 = 'Spare' | German: 'S1_Prompts German 929' | French: 'S1_Prompts French 929'
  930 = 'Waiting for Clamp Cylinder A1 Advance... Check Q1.0...' | German: 'S1_Prompts German 930' | French: 'S1_Prompts French 930'
  931 = 'Waiting for Clamp Cylinder A1 Return... Check Q1.1...' | German: 'S1_Prompts German 931' | French: 'S1_Prompts French 931'
  932 = 'Spare' | German: 'S1_Prompts German 932' | French: 'S1_Prompts French 932'
  933 = 'Spare' | German: 'S1_Prompts German 933' | French: 'S1_Prompts French 933'
  934 = 'Spare' | German: 'S1_Prompts German 934' | French: 'S1_Prompts French 934'
  935 = 'Spare' | German: 'S1_Prompts German 935' | French: 'S1_Prompts French 935'
  936 = 'Spare' | German: 'S1_Prompts German 936' | French: 'S1_Prompts French 936'
  937 = 'Spare' | German: 'S1_Prompts German 937' | French: 'S1_Prompts French 937'
  938 = 'Spare' | German: 'S1_Prompts German 938' | French: 'S1_Prompts French 938'
  939 = 'Spare' | German: 'S1_Prompts German 939' | French: 'S1_Prompts French 939'
  940 = 'Waiting for Clamp Cylinder A1 Advance... Check Q1.0...' | German: 'S1_Prompts German 940' | French: 'S1_Prompts French 940'
  941 = 'Waiting for Clamp Cylinder A1 Return... Check Q1.1...' | German: 'S1_Prompts German 941' | French: 'S1_Prompts French 941'
  942 = 'Spare' | German: 'S1_Prompts German 942' | French: 'S1_Prompts French 942'
  943 = 'Spare' | German: 'S1_Prompts German 943' | French: 'S1_Prompts French 943'
  944 = 'Spare' | German: 'S1_Prompts German 944' | French: 'S1_Prompts French 944'
  945 = 'Spare' | German: 'S1_Prompts German 945' | French: 'S1_Prompts French 945'
  946 = 'Spare' | German: 'S1_Prompts German 946' | French: 'S1_Prompts French 946'
  947 = 'Spare' | German: 'S1_Prompts German 947' | French: 'S1_Prompts French 947'
  948 = 'Spare' | German: 'S1_Prompts German 948' | French: 'S1_Prompts French 948'
  949 = 'Spare' | German: 'S1_Prompts German 949' | French: 'S1_Prompts French 949'
  950 = 'Waiting for Clamp Cylinder A1 Advance... Check Q1.0...' | German: 'S1_Prompts German 950' | French: 'S1_Prompts French 950'
  951 = 'Waiting for Clamp Cylinder A1 Return... Check Q1.1...' | German: 'S1_Prompts German 951' | French: 'S1_Prompts French 951'
  952 = 'Spare' | German: 'S1_Prompts German 952' | French: 'S1_Prompts French 952'
  953 = 'Spare' | German: 'S1_Prompts German 953' | French: 'S1_Prompts French 953'
  954 = 'Spare' | German: 'S1_Prompts German 954' | French: 'S1_Prompts French 954'
  955 = 'Spare' | German: 'S1_Prompts German 955' | French: 'S1_Prompts French 955'
  956 = 'Spare' | German: 'S1_Prompts German 956' | French: 'S1_Prompts French 956'
  957 = 'Spare' | German: 'S1_Prompts German 957' | French: 'S1_Prompts French 957'
  958 = 'Spare' | German: 'S1_Prompts German 958' | French: 'S1_Prompts French 958'
  959 = 'Spare' | German: 'S1_Prompts German 959' | French: 'S1_Prompts French 959'
  960 = 'Waiting for Clamp Cylinder A1 Advance... Check Q1.0...' | German: 'S1_Prompts German 960' | French: 'S1_Prompts French 960'
  961 = 'Waiting for Clamp Cylinder A1 Return... Check Q1.1...' | German: 'S1_Prompts German 961' | French: 'S1_Prompts French 961'
  962 = 'Spare' | German: 'S1_Prompts German 962' | French: 'S1_Prompts French 962'
  963 = 'Spare' | German: 'S1_Prompts German 963' | French: 'S1_Prompts French 963'
  964 = 'Spare' | German: 'S1_Prompts German 964' | French: 'S1_Prompts French 964'
  965 = 'Spare' | German: 'S1_Prompts German 965' | French: 'S1_Prompts French 965'
  966 = 'Spare' | German: 'S1_Prompts German 966' | French: 'S1_Prompts French 966'
  967 = 'Spare' | German: 'S1_Prompts German 967' | French: 'S1_Prompts French 967'
  968 = 'Spare' | German: 'S1_Prompts German 968' | French: 'S1_Prompts French 968'
  969 = 'Spare' | German: 'S1_Prompts German 969' | French: 'S1_Prompts French 969'
  970 = 'Waiting for Clamp Cylinder A1 Advance... Check Q1.0...' | German: 'S1_Prompts German 970' | French: 'S1_Prompts French 970'
  971 = 'Waiting for Clamp Cylinder A1 Return... Check Q1.1...' | German: 'S1_Prompts German 971' | French: 'S1_Prompts French 971'
  972 = 'Spare' | German: 'S1_Prompts German 972' | French: 'S1_Prompts French 972'
  973 = 'Spare' | German: 'S1_Prompts German 973' | French: 'S1_Prompts French 973'
  974 = 'Spare' | German: 'S1_Prompts German 974' | French: 'S1_Prompts French 974'
  975 = 'Spare' | German: 'S1_Prompts German 975' | French: 'S1_Prompts French 975'
  976 = 'Spare' | German: 'S1_Prompts German 976' | French: 'S1_Prompts French 976'
  977 = 'Spare' | German: 'S1_Prompts German 977' | French: 'S1_Prompts French 977'
  978 = 'Spare' | German: 'S1_Prompts German 978' | French: 'S1_Prompts French 978'
  979 = 'Spare' | German: 'S1_Prompts German 979' | French: 'S1_Prompts French 979'
  980 = 'Waiting for End of Station 1 A1 Advance... Check Q1.0...' | German: 'S1_Prompts German 980' | French: 'S1_Prompts French 980'
  981 = 'Waiting for End of Station 1 A1 Return... Check Q1.1...' | German: 'S1_Prompts German 981' | French: 'S1_Prompts French 981'
  982 = 'Spare' | German: 'S1_Prompts German 982' | French: 'S1_Prompts French 982'
  983 = 'Spare' | German: 'S1_Prompts German 983' | French: 'S1_Prompts French 983'
  984 = 'Spare' | German: 'S1_Prompts German 984' | French: 'S1_Prompts French 984'
  985 = 'Spare' | German: 'S1_Prompts German 985' | French: 'S1_Prompts French 985'
  986 = 'Spare' | German: 'S1_Prompts German 986' | French: 'S1_Prompts French 986'
  987 = 'Spare' | German: 'S1_Prompts German 987' | French: 'S1_Prompts French 987'
  988 = 'Spare' | German: 'S1_Prompts German 988' | French: 'S1_Prompts French 988'
  989 = 'Spare' | German: 'S1_Prompts German 989' | French: 'S1_Prompts French 989'
  990 = 'S1_Prompts Default 990' | German: 'S1_Prompts German 990' | French: 'S1_Prompts French 990'
  991 = 'S1_Prompts Default 991' | German: 'S1_Prompts German 991' | French: 'S1_Prompts French 991'
  992 = 'S1_Prompts Default 992' | German: 'S1_Prompts German 992' | French: 'S1_Prompts French 992'
  993 = 'S1_Prompts Default 993' | German: 'S1_Prompts German 993' | French: 'S1_Prompts French 993'
  994 = 'S1_Prompts Default 994' | German: 'S1_Prompts German 994' | French: 'S1_Prompts French 994'
  995 = 'S1_Prompts Default 995' | German: 'S1_Prompts German 995' | French: 'S1_Prompts French 995'
  996 = 'S1_Prompts Default 996' | German: 'S1_Prompts German 996' | French: 'S1_Prompts French 996'
  997 = 'S1_Prompts Default 997' | German: 'S1_Prompts German 997' | French: 'S1_Prompts French 997'
  998 = 'S1_Prompts Default 998' | German: 'S1_Prompts German 998' | French: 'S1_Prompts French 998'
  999 = 'S1_Prompts Default 999' | German: 'S1_Prompts German 999' | French: 'S1_Prompts French 999'
  1000 = 'S1_Prompts Default 1000' | German: 'S1_Prompts German 1000' | French: 'S1_Prompts French 1000'
   = ''
END_TEXTLIST

(* stored: Version 1.1.0.1, ProductVersion 3.1.4024.12
   TextList S1_Prompts: Id {18e589f1-43d4-40ee-8eaf-6df4fa95381b} *)
